// LS Electric XG5000 project: X3353 JOSUNG UPDATE
// PLC NewPLC
// module base 0 slot 0: Motion Module:XGF-M32E (EtherCAT Network, 32-Axis)
// module base 0 slot 1: Input Module:XGI-D28A/B (DC 24V Input, 64 Contacts)
// module base 0 slot 2: Input Module:XGI-D28A/B (DC 24V Input, 64 Contacts)
// module base 0 slot 3: Output Module:XGQ-TR8A/B (Transistor Output, 64 Contacts (0.1A, Sink Output/Source Output))
// module base 0 slot 4: Output Module:XGQ-TR8A/B (Transistor Output, 64 Contacts (0.1A, Sink Output/Source Output))
// module base 0 slot 5: Analog Input Module:XGF-AD16A (A/D Voltage/Current Input Type(16 Channels))
// module base 0 slot 6: Analog Input Module:XGF-AD16A (A/D Voltage/Current Input Type(16 Channels))
// module base 0 slot 7: FEnet:XGL-EFMT(B) (Fast Ethernet Module, Electrical Master)
// module base 0 slot 8: FEnet:XGL-EFMT(B) (Fast Ethernet Module, Electrical Master)

PROGRAM 01_MAIN (task: ¨ö¨¬A¥ì CA¡¤I¡¾¡¿¡¤¡Í)

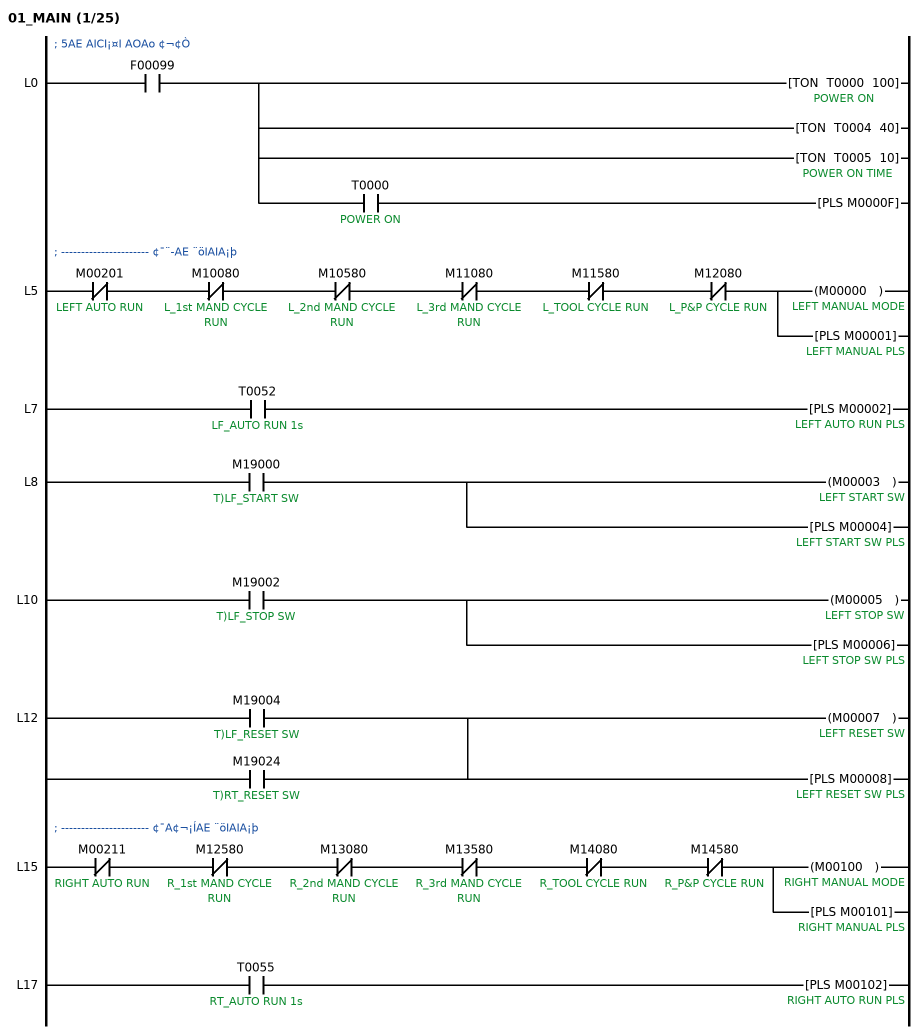
; L0
LOAD      F00099
TON       T0000 100	// POWER ON
TON       T0004 40
TON       T0005 10	// POWER ON TIME
AND       T0000	// POWER ON
OUTP      M0000F
// output comment: 5AE AICI¡¤I AOAo ¢¬¢Ò
// ---------------------- ¢¯¨­AE ¨öIAIA¡þ
; L5
LOAD NOT  M00201	// LEFT AUTO RUN
AND NOT   M10080	// L_1st MAND CYCLE RUN
AND NOT   M10580	// L_2nd MAND CYCLE RUN
AND NOT   M11080	// L_3rd MAND CYCLE RUN
AND NOT   M11580	// L_TOOL CYCLE RUN
AND NOT   M12080	// L_P&P CYCLE RUN
OUT       M00000	// LEFT MANUAL MODE
OUTP      M00001	// LEFT MANUAL PLS
; L7
LOAD      T0052	// LF_AUTO RUN 1s
OUTP      M00002	// LEFT AUTO RUN PLS
; L8
LOAD      M19000	// T)LF_START SW
OUT       M00003	// LEFT START SW
OUTP      M00004	// LEFT START SW PLS
; L10
LOAD      M19002	// T)LF_STOP SW
OUT       M00005	// LEFT STOP SW
OUTP      M00006	// LEFT STOP SW PLS
; L12
LOAD      M19004	// T)LF_RESET SW
OR        M19024	// T)RT_RESET SW
OUT       M00007	// LEFT RESET SW
OUTP      M00008	// LEFT RESET SW PLS
// ---------------------- ¢¯A¢¬¡ÍAE ¨öIAIA¡þ
; L15
LOAD NOT  M00211	// RIGHT AUTO RUN
AND NOT   M12580	// R_1st MAND CYCLE RUN
AND NOT   M13080	// R_2nd MAND CYCLE RUN
AND NOT   M13580	// R_3rd MAND CYCLE RUN
AND NOT   M14080	// R_TOOL CYCLE RUN
AND NOT   M14580	// R_P&P CYCLE RUN
OUT       M00100	// RIGHT MANUAL MODE
OUTP      M00101	// RIGHT MANUAL PLS
; L17
LOAD      T0055	// RT_AUTO RUN 1s
OUTP      M00102	// RIGHT AUTO RUN PLS

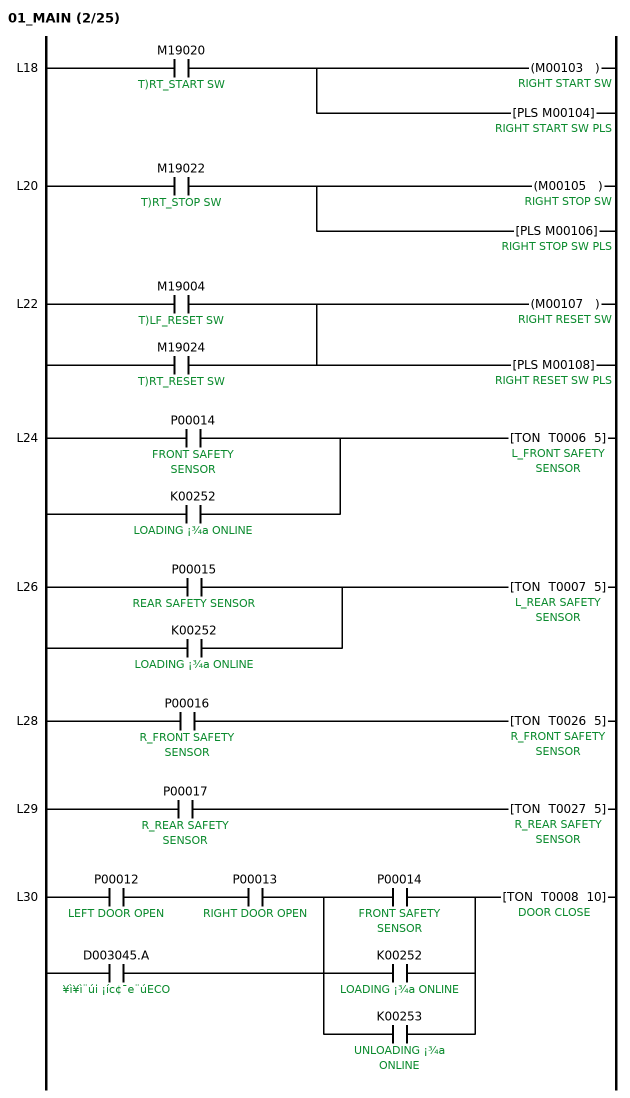
; L18
LOAD      M19020	// T)RT_START SW
OUT       M00103	// RIGHT START SW
OUTP      M00104	// RIGHT START SW PLS
; L20
LOAD      M19022	// T)RT_STOP SW
OUT       M00105	// RIGHT STOP SW
OUTP      M00106	// RIGHT STOP SW PLS
; L22
LOAD      M19004	// T)LF_RESET SW
OR        M19024	// T)RT_RESET SW
OUT       M00107	// RIGHT RESET SW
OUTP      M00108	// RIGHT RESET SW PLS
; L24
LOAD      P00014	// FRONT SAFETY SENSOR
OR        K00252	// LOADING ¡¾a ONLINE
TON       T0006 5	// L_FRONT SAFETY SENSOR
; L26
LOAD      P00015	// REAR SAFETY SENSOR
OR        K00252	// LOADING ¡¾a ONLINE
TON       T0007 5	// L_REAR SAFETY SENSOR
; L28
LOAD      P00016	// R_FRONT SAFETY SENSOR
TON       T0026 5	// R_FRONT SAFETY SENSOR
; L29
LOAD      P00017	// R_REAR SAFETY SENSOR
TON       T0027 5	// R_REAR SAFETY SENSOR
; L30
LOAD      P00012	// LEFT DOOR OPEN
AND       P00013	// RIGHT DOOR OPEN
OR        D003045.A	// ¥ì¥ì¨úi ¡íc¢¯e¨úECO
LOAD      P00014	// FRONT SAFETY SENSOR
OR        K00252	// LOADING ¡¾a ONLINE
OR        K00253	// UNLOADING ¡¾a ONLINE
AND LOAD
TON       T0008 10	// DOOR CLOSE

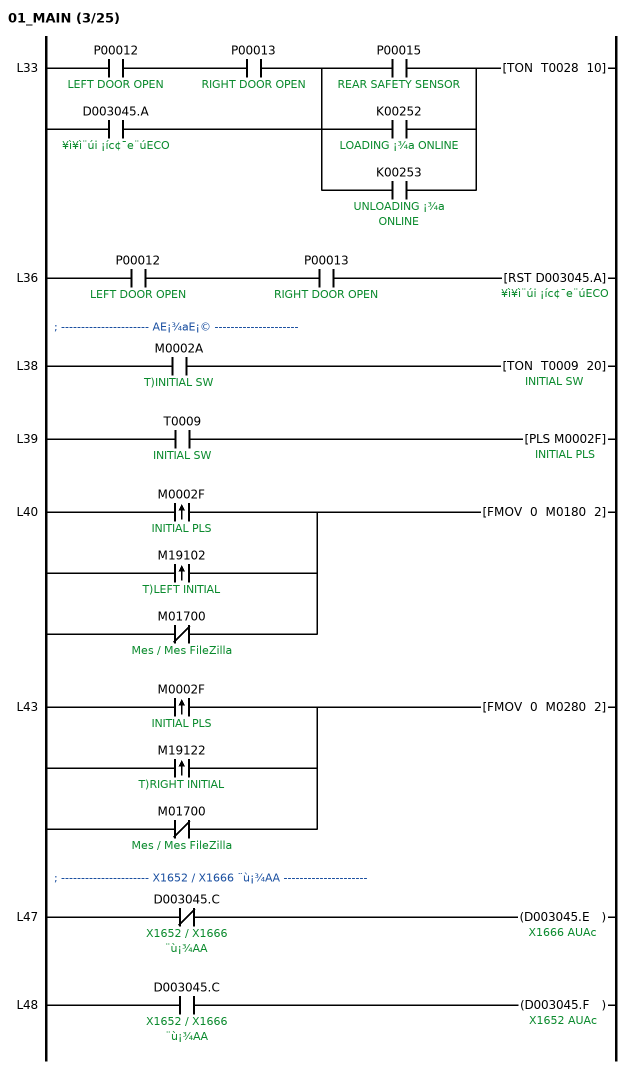
; L33
LOAD      P00012	// LEFT DOOR OPEN
AND       P00013	// RIGHT DOOR OPEN
OR        D003045.A	// ¥ì¥ì¨úi ¡íc¢¯e¨úECO
LOAD      P00015	// REAR SAFETY SENSOR
OR        K00252	// LOADING ¡¾a ONLINE
OR        K00253	// UNLOADING ¡¾a ONLINE
AND LOAD
TON       T0028 10
; L36
LOAD      P00012	// LEFT DOOR OPEN
AND       P00013	// RIGHT DOOR OPEN
RST       D003045.A	// ¥ì¥ì¨úi ¡íc¢¯e¨úECO
// ---------------------- AE¡¾aE¡© ---------------------
; L38
LOAD      M0002A	// T)INITIAL SW
TON       T0009 20	// INITIAL SW
; L39
LOAD      T0009	// INITIAL SW
OUTP      M0002F	// INITIAL PLS
; L40
LOADP     M0002F	// INITIAL PLS
ORP       M19102	// T)LEFT INITIAL
OR NOT    M01700	// Mes / Mes FileZilla
FMOV      0 M0180 2
; L43
LOADP     M0002F	// INITIAL PLS
ORP       M19122	// T)RIGHT INITIAL
OR NOT    M01700	// Mes / Mes FileZilla
FMOV      0 M0280 2
// ---------------------- X1652 / X1666 ¨ù¡¾AA ---------------------
; L47
LOAD NOT  D003045.C	// X1652 / X1666 ¨ù¡¾AA
OUT       D003045.E	// X1666 AUAc
; L48
LOAD      D003045.C	// X1652 / X1666 ¨ù¡¾AA
OUT       D003045.F	// X1652 AUAc

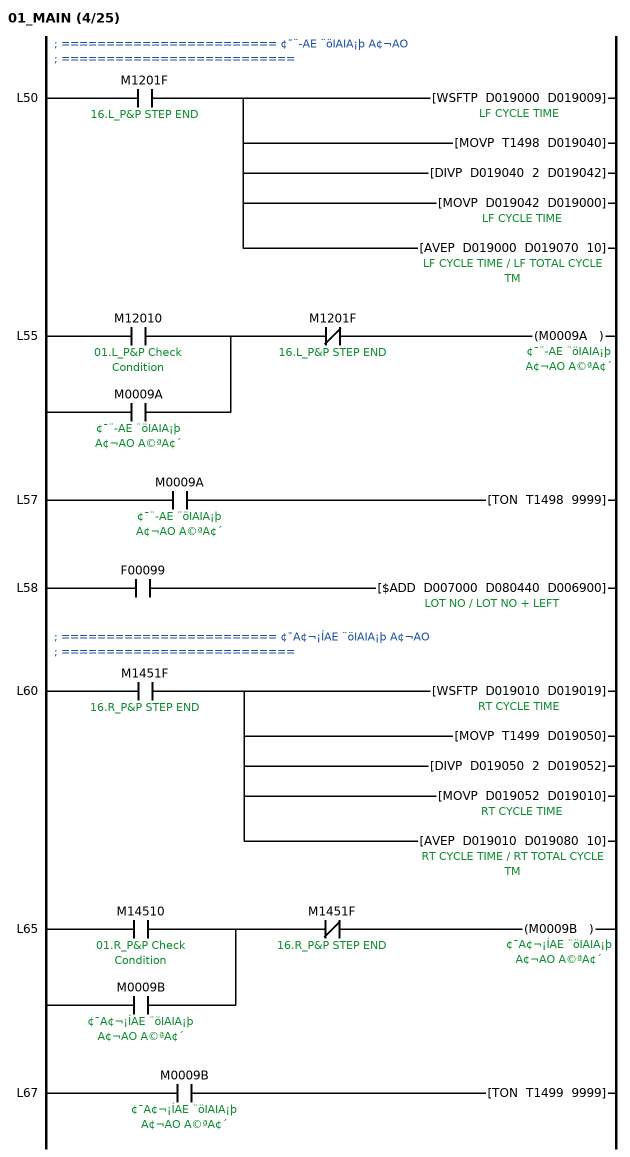
// ======================== ¢¯¨­AE ¨öIAIA¡þ A¢¬AO ==========================
; L50
LOAD      M1201F	// 16.L_P&P STEP END
WSFTP     D019000 D019009	// LF CYCLE TIME
MOVP      T1498 D019040
DIVP      D019040 2 D019042
MOVP      D019042 D019000	// LF CYCLE TIME
AVEP      D019000 D019070 10	// LF CYCLE TIME / LF TOTAL CYCLE TM
; L55
LOAD      M12010	// 01.L_P&P Check Condition
OR        M0009A	// ¢¯¨­AE ¨öIAIA¡þ A¢¬AO A©ªA¢´
AND NOT   M1201F	// 16.L_P&P STEP END
OUT       M0009A	// ¢¯¨­AE ¨öIAIA¡þ A¢¬AO A©ªA¢´
; L57
LOAD      M0009A	// ¢¯¨­AE ¨öIAIA¡þ A¢¬AO A©ªA¢´
TON       T1498 9999
; L58
LOAD      F00099
$ADD      D007000 D080440 D006900	// LOT NO / LOT NO + LEFT
// ======================== ¢¯A¢¬¡ÍAE ¨öIAIA¡þ A¢¬AO ==========================
; L60
LOAD      M1451F	// 16.R_P&P STEP END
WSFTP     D019010 D019019	// RT CYCLE TIME
MOVP      T1499 D019050
DIVP      D019050 2 D019052
MOVP      D019052 D019010	// RT CYCLE TIME
AVEP      D019010 D019080 10	// RT CYCLE TIME / RT TOTAL CYCLE TM
; L65
LOAD      M14510	// 01.R_P&P Check Condition
OR        M0009B	// ¢¯A¢¬¡ÍAE ¨öIAIA¡þ A¢¬AO A©ªA¢´
AND NOT   M1451F	// 16.R_P&P STEP END
OUT       M0009B	// ¢¯A¢¬¡ÍAE ¨öIAIA¡þ A¢¬AO A©ªA¢´
; L67
LOAD      M0009B	// ¢¯A¢¬¡ÍAE ¨öIAIA¡þ A¢¬AO A©ªA¢´
TON       T1499 9999

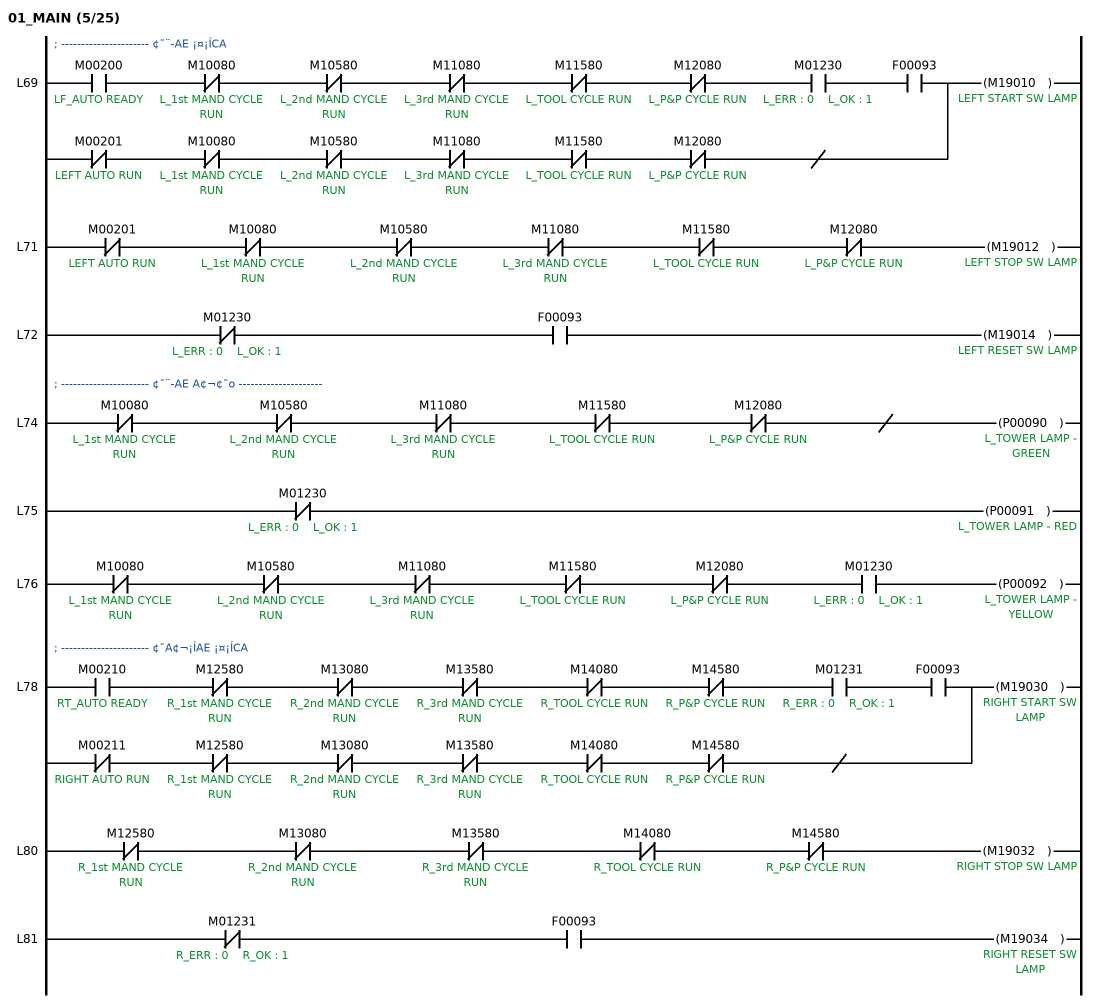
// ---------------------- ¢¯¨­AE ¡¤¡ÍCA
; L69
LOAD      M00200	// LF_AUTO READY
AND NOT   M10080	// L_1st MAND CYCLE RUN
AND NOT   M10580	// L_2nd MAND CYCLE RUN
AND NOT   M11080	// L_3rd MAND CYCLE RUN
AND NOT   M11580	// L_TOOL CYCLE RUN
AND NOT   M12080	// L_P&P CYCLE RUN
AND       M01230	// L_ERR : 0    L_OK : 1
AND       F00093
LOAD NOT  M00201	// LEFT AUTO RUN
AND NOT   M10080	// L_1st MAND CYCLE RUN
AND NOT   M10580	// L_2nd MAND CYCLE RUN
AND NOT   M11080	// L_3rd MAND CYCLE RUN
AND NOT   M11580	// L_TOOL CYCLE RUN
AND NOT   M12080	// L_P&P CYCLE RUN
NOT
OR LOAD
OUT       M19010	// LEFT START SW LAMP
; L71
LOAD NOT  M00201	// LEFT AUTO RUN
AND NOT   M10080	// L_1st MAND CYCLE RUN
AND NOT   M10580	// L_2nd MAND CYCLE RUN
AND NOT   M11080	// L_3rd MAND CYCLE RUN
AND NOT   M11580	// L_TOOL CYCLE RUN
AND NOT   M12080	// L_P&P CYCLE RUN
OUT       M19012	// LEFT STOP SW LAMP
; L72
LOAD NOT  M01230	// L_ERR : 0    L_OK : 1
AND       F00093
OUT       M19014	// LEFT RESET SW LAMP
// ---------------------- ¢¯¨­AE A¢¬¢¯o ---------------------
; L74
LOAD NOT  M10080	// L_1st MAND CYCLE RUN
AND NOT   M10580	// L_2nd MAND CYCLE RUN
AND NOT   M11080	// L_3rd MAND CYCLE RUN
AND NOT   M11580	// L_TOOL CYCLE RUN
AND NOT   M12080	// L_P&P CYCLE RUN
NOT
OUT       P00090	// L_TOWER LAMP - GREEN
; L75
LOAD NOT  M01230	// L_ERR : 0    L_OK : 1
OUT       P00091	// L_TOWER LAMP - RED
; L76
LOAD NOT  M10080	// L_1st MAND CYCLE RUN
AND NOT   M10580	// L_2nd MAND CYCLE RUN
AND NOT   M11080	// L_3rd MAND CYCLE RUN
AND NOT   M11580	// L_TOOL CYCLE RUN
AND NOT   M12080	// L_P&P CYCLE RUN
AND       M01230	// L_ERR : 0    L_OK : 1
OUT       P00092	// L_TOWER LAMP - YELLOW
// ---------------------- ¢¯A¢¬¡ÍAE ¡¤¡ÍCA
; L78
LOAD      M00210	// RT_AUTO READY
AND NOT   M12580	// R_1st MAND CYCLE RUN
AND NOT   M13080	// R_2nd MAND CYCLE RUN
AND NOT   M13580	// R_3rd MAND CYCLE RUN
AND NOT   M14080	// R_TOOL CYCLE RUN
AND NOT   M14580	// R_P&P CYCLE RUN
AND       M01231	// R_ERR : 0    R_OK : 1
AND       F00093
LOAD NOT  M00211	// RIGHT AUTO RUN
AND NOT   M12580	// R_1st MAND CYCLE RUN
AND NOT   M13080	// R_2nd MAND CYCLE RUN
AND NOT   M13580	// R_3rd MAND CYCLE RUN
AND NOT   M14080	// R_TOOL CYCLE RUN
AND NOT   M14580	// R_P&P CYCLE RUN
NOT
OR LOAD
OUT       M19030	// RIGHT START SW LAMP
; L80
LOAD NOT  M12580	// R_1st MAND CYCLE RUN
AND NOT   M13080	// R_2nd MAND CYCLE RUN
AND NOT   M13580	// R_3rd MAND CYCLE RUN
AND NOT   M14080	// R_TOOL CYCLE RUN
AND NOT   M14580	// R_P&P CYCLE RUN
OUT       M19032	// RIGHT STOP SW LAMP
; L81
LOAD NOT  M01231	// R_ERR : 0    R_OK : 1
AND       F00093
OUT       M19034	// RIGHT RESET SW LAMP

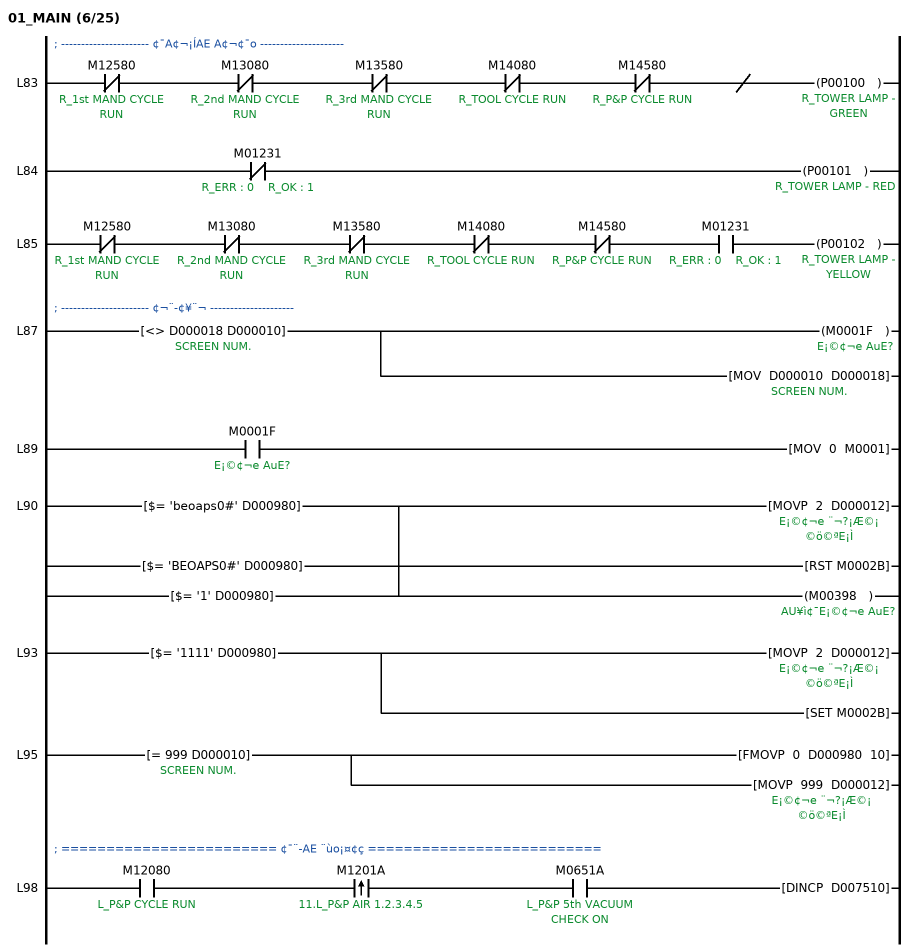
// ---------------------- ¢¯A¢¬¡ÍAE A¢¬¢¯o ---------------------
; L83
LOAD NOT  M12580	// R_1st MAND CYCLE RUN
AND NOT   M13080	// R_2nd MAND CYCLE RUN
AND NOT   M13580	// R_3rd MAND CYCLE RUN
AND NOT   M14080	// R_TOOL CYCLE RUN
AND NOT   M14580	// R_P&P CYCLE RUN
NOT
OUT       P00100	// R_TOWER LAMP - GREEN
; L84
LOAD NOT  M01231	// R_ERR : 0    R_OK : 1
OUT       P00101	// R_TOWER LAMP - RED
; L85
LOAD NOT  M12580	// R_1st MAND CYCLE RUN
AND NOT   M13080	// R_2nd MAND CYCLE RUN
AND NOT   M13580	// R_3rd MAND CYCLE RUN
AND NOT   M14080	// R_TOOL CYCLE RUN
AND NOT   M14580	// R_P&P CYCLE RUN
AND       M01231	// R_ERR : 0    R_OK : 1
OUT       P00102	// R_TOWER LAMP - YELLOW
// ---------------------- ¢¬¨­¢¥¨¬ ---------------------
; L87
LOAD<>    D000018 D000010	// SCREEN NUM.
OUT       M0001F	// E¡©¢¬e AuE?
MOV       D000010 D000018	// SCREEN NUM.
; L89
LOAD      M0001F	// E¡©¢¬e AuE?
MOV       0 M0001
; L90
LOAD$=    'beoaps0#' D000980
OR$=      'BEOAPS0#' D000980
OR$=      '1' D000980
MOVP      2 D000012	// E¡©¢¬e ¨¬?¡Æ©¡ ©ö©ªE¡Ì
RST       M0002B
OUT       M00398	// AU¥ì¢¯E¡©¢¬e AuE?
; L93
LOAD$=    '1111' D000980
MOVP      2 D000012	// E¡©¢¬e ¨¬?¡Æ©¡ ©ö©ªE¡Ì
SET       M0002B
; L95
LOAD=     999 D000010	// SCREEN NUM.
FMOVP     0 D000980 10
MOVP      999 D000012	// E¡©¢¬e ¨¬?¡Æ©¡ ©ö©ªE¡Ì
// ======================== ¢¯¨­AE ¨ùo¡¤¢ç ==========================
; L98
LOAD      M12080	// L_P&P CYCLE RUN
ANDP      M1201A	// 11.L_P&P AIR 1.2.3.4.5
AND       M0651A	// L_P&P 5th VACUUM CHECK ON
DINCP     D007510

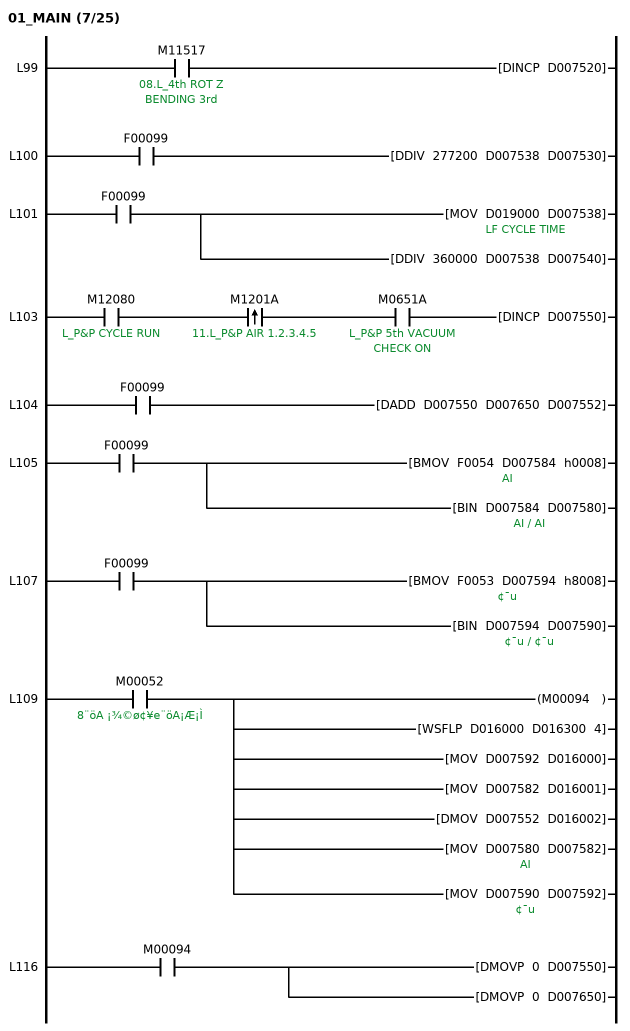
; L99
LOAD      M11517	// 08.L_4th ROT Z BENDING 3rd
DINCP     D007520
; L100
LOAD      F00099
DDIV      277200 D007538 D007530
; L101
LOAD      F00099
MOV       D019000 D007538	// LF CYCLE TIME
DDIV      360000 D007538 D007540
; L103
LOAD      M12080	// L_P&P CYCLE RUN
ANDP      M1201A	// 11.L_P&P AIR 1.2.3.4.5
AND       M0651A	// L_P&P 5th VACUUM CHECK ON
DINCP     D007550
; L104
LOAD      F00099
DADD      D007550 D007650 D007552
; L105
LOAD      F00099
BMOV      F0054 D007584 h0008	// AI
BIN       D007584 D007580	// AI / AI
; L107
LOAD      F00099
BMOV      F0053 D007594 h8008	// ¢¯u
BIN       D007594 D007590	// ¢¯u / ¢¯u
; L109
LOAD      M00052	// 8¨öA ¡¾©ø¢¥e¨öA¡Æ¡Ì
OUT       M00094
WSFLP     D016000 D016300 4
MOV       D007592 D016000
MOV       D007582 D016001
DMOV      D007552 D016002
MOV       D007580 D007582	// AI
MOV       D007590 D007592	// ¢¯u
; L116
LOAD      M00094
DMOVP     0 D007550
DMOVP     0 D007650

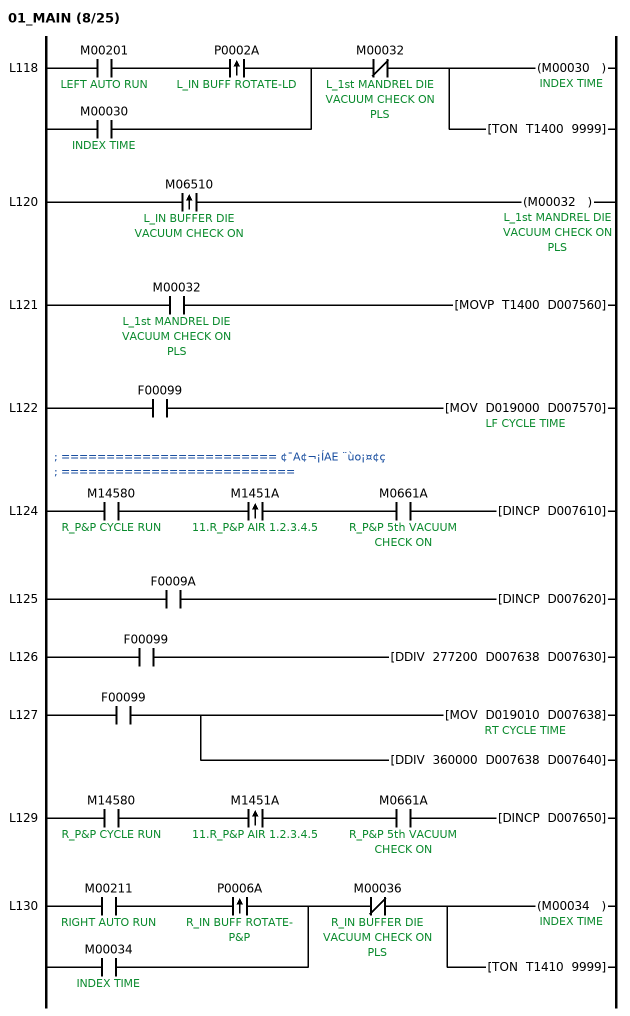
; L118
LOAD      M00201	// LEFT AUTO RUN
ANDP      P0002A	// L_IN BUFF ROTATE-LD
OR        M00030	// INDEX TIME
AND NOT   M00032	// L_1st MANDREL DIE VACUUM CHECK ON PLS
OUT       M00030	// INDEX TIME
TON       T1400 9999
; L120
LOADP     M06510	// L_IN BUFFER DIE VACUUM CHECK ON
OUT       M00032	// L_1st MANDREL DIE VACUUM CHECK ON PLS
; L121
LOAD      M00032	// L_1st MANDREL DIE VACUUM CHECK ON PLS
MOVP      T1400 D007560
; L122
LOAD      F00099
MOV       D019000 D007570	// LF CYCLE TIME
// ======================== ¢¯A¢¬¡ÍAE ¨ùo¡¤¢ç ==========================
; L124
LOAD      M14580	// R_P&P CYCLE RUN
ANDP      M1451A	// 11.R_P&P AIR 1.2.3.4.5
AND       M0661A	// R_P&P 5th VACUUM CHECK ON
DINCP     D007610
; L125
LOAD      F0009A
DINCP     D007620
; L126
LOAD      F00099
DDIV      277200 D007638 D007630
; L127
LOAD      F00099
MOV       D019010 D007638	// RT CYCLE TIME
DDIV      360000 D007638 D007640
; L129
LOAD      M14580	// R_P&P CYCLE RUN
ANDP      M1451A	// 11.R_P&P AIR 1.2.3.4.5
AND       M0661A	// R_P&P 5th VACUUM CHECK ON
DINCP     D007650
; L130
LOAD      M00211	// RIGHT AUTO RUN
ANDP      P0006A	// R_IN BUFF ROTATE- P&P
OR        M00034	// INDEX TIME
AND NOT   M00036	// R_IN BUFFER DIE VACUUM CHECK ON PLS
OUT       M00034	// INDEX TIME
TON       T1410 9999

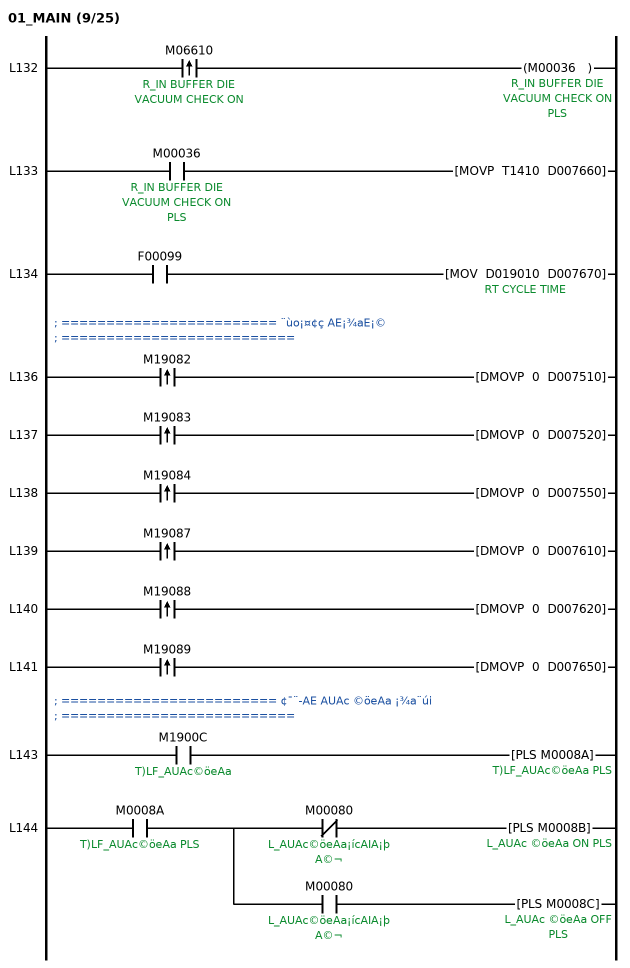
; L132
LOADP     M06610	// R_IN BUFFER DIE VACUUM CHECK ON
OUT       M00036	// R_IN BUFFER DIE VACUUM CHECK ON PLS
; L133
LOAD      M00036	// R_IN BUFFER DIE VACUUM CHECK ON PLS
MOVP      T1410 D007660
; L134
LOAD      F00099
MOV       D019010 D007670	// RT CYCLE TIME
// ======================== ¨ùo¡¤¢ç AE¡¾aE¡© ==========================
; L136
LOADP     M19082
DMOVP     0 D007510
; L137
LOADP     M19083
DMOVP     0 D007520
; L138
LOADP     M19084
DMOVP     0 D007550
; L139
LOADP     M19087
DMOVP     0 D007610
; L140
LOADP     M19088
DMOVP     0 D007620
; L141
LOADP     M19089
DMOVP     0 D007650
// ======================== ¢¯¨­AE AUAc ©öeAa ¡¾a¨úi ==========================
; L143
LOAD      M1900C	// T)LF_AUAc©öeAa
OUTP      M0008A	// T)LF_AUAc©öeAa PLS
; L144
LOAD      M0008A	// T)LF_AUAc©öeAa PLS
MPUSH
AND NOT   M00080	// L_AUAc©öeAa¡ícAIA¡þA©¬
OUTP      M0008B	// L_AUAc ©öeAa ON PLS
MPOP
AND       M00080	// L_AUAc©öeAa¡ícAIA¡þA©¬
OUTP      M0008C	// L_AUAc ©öeAa OFF PLS

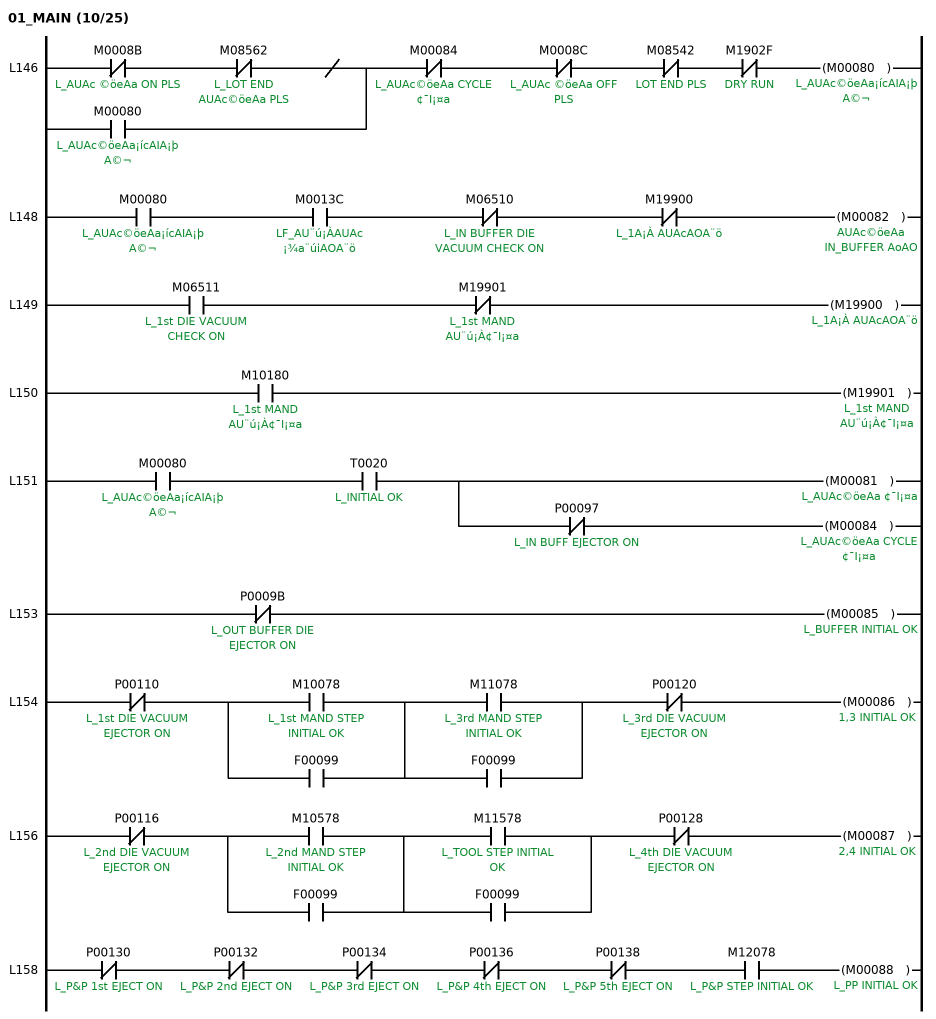
; L146
LOAD NOT  M0008B	// L_AUAc ©öeAa ON PLS
AND NOT   M08562	// L_LOT END AUAc©öeAa PLS
NOT
OR        M00080	// L_AUAc©öeAa¡ícAIA¡þA©¬
AND NOT   M00084	// L_AUAc©öeAa CYCLE ¢¯I¡¤a
AND NOT   M0008C	// L_AUAc ©öeAa OFF PLS
AND NOT   M08542	// LOT END PLS
AND NOT   M1902F	// DRY RUN
OUT       M00080	// L_AUAc©öeAa¡ícAIA¡þA©¬
; L148
LOAD      M00080	// L_AUAc©öeAa¡ícAIA¡þA©¬
AND       M0013C	// LF_AU¨ú¡ÀAUAc ¡¾a¨úiAOA¨ö
AND NOT   M06510	// L_IN BUFFER DIE VACUUM CHECK ON
AND NOT   M19900	// L_1A¡À AUAcAOA¨ö
OUT       M00082	// AUAc©öeAa IN_BUFFER AoAO 
; L149
LOAD      M06511	// L_1st DIE VACUUM CHECK ON
AND NOT   M19901	// L_1st MAND AU¨ú¡À¢¯I¡¤a
OUT       M19900	// L_1A¡À AUAcAOA¨ö
; L150
LOAD      M10180	// L_1st MAND AU¨ú¡À¢¯I¡¤a
OUT       M19901	// L_1st MAND AU¨ú¡À¢¯I¡¤a
; L151
LOAD      M00080	// L_AUAc©öeAa¡ícAIA¡þA©¬
AND       T0020	// L_INITIAL OK
OUT       M00081	// L_AUAc©öeAa ¢¯I¡¤a
AND NOT   P00097	// L_IN BUFF EJECTOR ON
OUT       M00084	// L_AUAc©öeAa CYCLE ¢¯I¡¤a
; L153
LOAD NOT  P0009B	// L_OUT BUFFER DIE EJECTOR ON
OUT       M00085	// L_BUFFER INITIAL OK
; L154
LOAD NOT  P00110	// L_1st DIE VACUUM EJECTOR ON
LOAD      M10078	// L_1st MAND STEP INITIAL OK
OR        F00099
AND LOAD
LOAD      M11078	// L_3rd MAND STEP INITIAL OK
OR        F00099
AND LOAD
AND NOT   P00120	// L_3rd DIE VACUUM EJECTOR ON
OUT       M00086	// 1,3 INITIAL OK
; L156
LOAD NOT  P00116	// L_2nd DIE VACUUM EJECTOR ON
LOAD      M10578	// L_2nd MAND STEP INITIAL OK
OR        F00099
AND LOAD
LOAD      M11578	// L_TOOL STEP INITIAL OK
OR        F00099
AND LOAD
AND NOT   P00128	// L_4th DIE VACUUM EJECTOR ON
OUT       M00087	// 2,4 INITIAL OK
; L158
LOAD NOT  P00130	// L_P&P 1st EJECT ON
AND NOT   P00132	// L_P&P 2nd EJECT ON
AND NOT   P00134	// L_P&P 3rd EJECT ON
AND NOT   P00136	// L_P&P 4th EJECT ON
AND NOT   P00138	// L_P&P 5th EJECT ON
AND       M12078	// L_P&P STEP INITIAL OK
OUT       M00088	// L_PP INITIAL OK

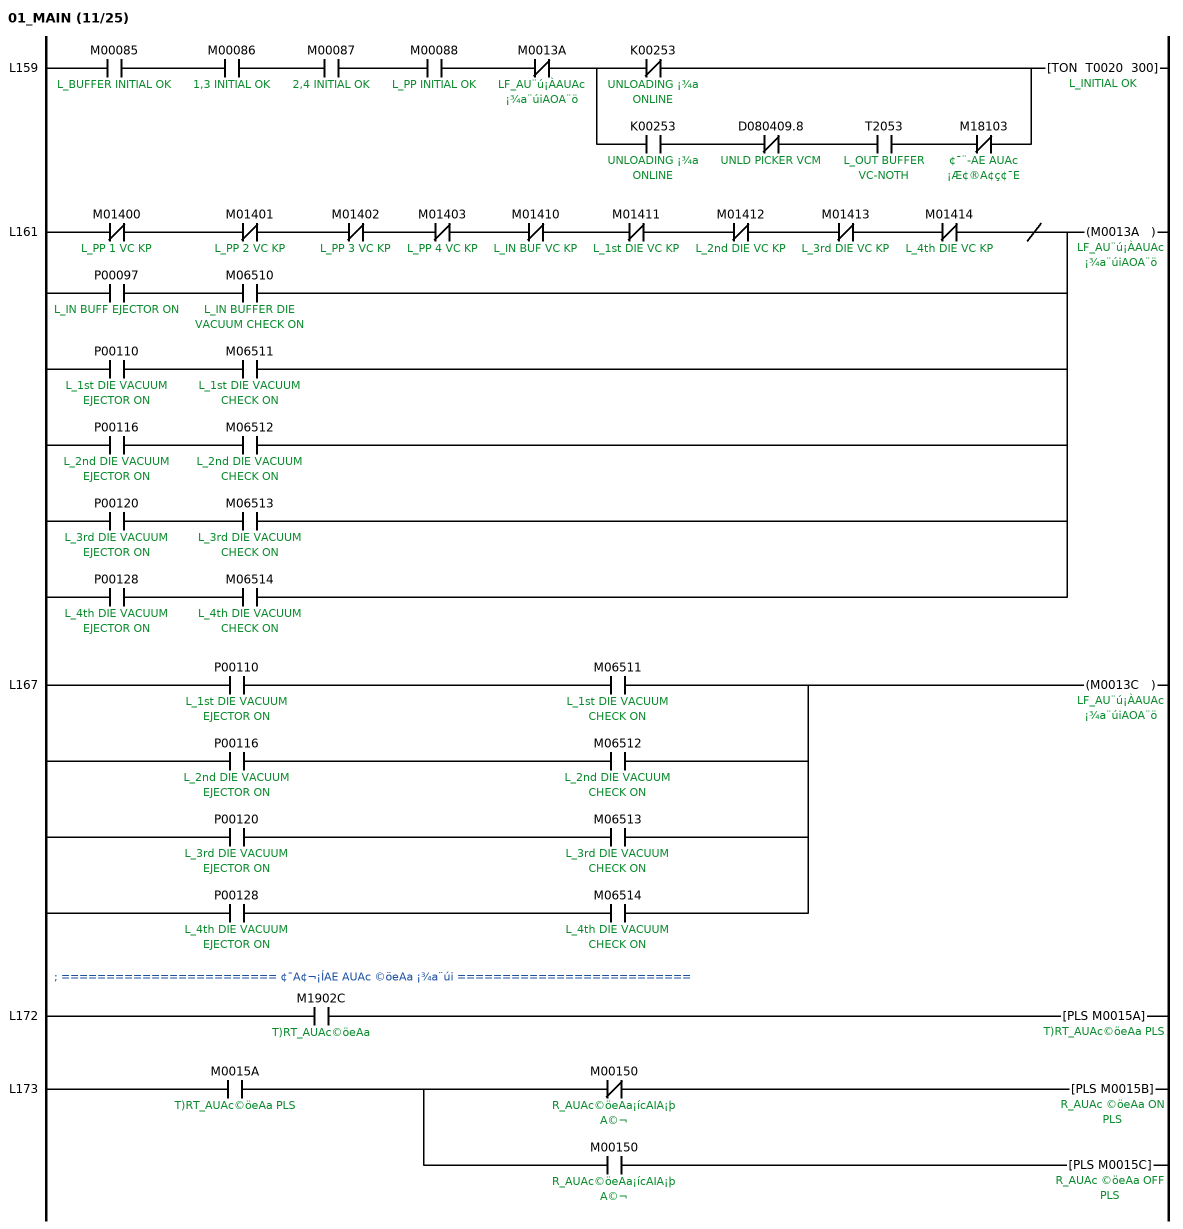
; L159
LOAD      M00085	// L_BUFFER INITIAL OK
AND       M00086	// 1,3 INITIAL OK
AND       M00087	// 2,4 INITIAL OK
AND       M00088	// L_PP INITIAL OK
AND NOT   M0013A	// LF_AU¨ú¡ÀAUAc ¡¾a¨úiAOA¨ö
LOAD NOT  K00253	// UNLOADING ¡¾a ONLINE
LOAD      K00253	// UNLOADING ¡¾a ONLINE
AND NOT   D080409.8	// UNLD PICKER VCM
AND       T2053	// L_OUT BUFFER VC-NOTH
AND NOT   M18103	// ¢¯¨­AE AUAc ¡Æ¢®A¢ç¢¯E
OR LOAD
AND LOAD
TON       T0020 300	// L_INITIAL OK
; L161
LOAD NOT  M01400	// L_PP 1 VC KP
AND NOT   M01401	// L_PP 2 VC KP
AND NOT   M01402	// L_PP 3 VC KP
AND NOT   M01403	// L_PP 4 VC KP
AND NOT   M01410	// L_IN BUF VC KP
AND NOT   M01411	// L_1st DIE VC KP
AND NOT   M01412	// L_2nd DIE VC KP
AND NOT   M01413	// L_3rd DIE VC KP
AND NOT   M01414	// L_4th DIE VC KP
NOT
LOAD      P00097	// L_IN BUFF EJECTOR ON
AND       M06510	// L_IN BUFFER DIE VACUUM CHECK ON
OR LOAD
LOAD      P00110	// L_1st DIE VACUUM EJECTOR ON
AND       M06511	// L_1st DIE VACUUM CHECK ON
OR LOAD
LOAD      P00116	// L_2nd DIE VACUUM EJECTOR ON
AND       M06512	// L_2nd DIE VACUUM CHECK ON
OR LOAD
LOAD      P00120	// L_3rd DIE VACUUM EJECTOR ON
AND       M06513	// L_3rd DIE VACUUM CHECK ON
OR LOAD
LOAD      P00128	// L_4th DIE VACUUM EJECTOR ON
AND       M06514	// L_4th DIE VACUUM CHECK ON
OR LOAD
OUT       M0013A	// LF_AU¨ú¡ÀAUAc ¡¾a¨úiAOA¨ö
; L167
LOAD      P00110	// L_1st DIE VACUUM EJECTOR ON
AND       M06511	// L_1st DIE VACUUM CHECK ON
LOAD      P00116	// L_2nd DIE VACUUM EJECTOR ON
AND       M06512	// L_2nd DIE VACUUM CHECK ON
OR LOAD
LOAD      P00120	// L_3rd DIE VACUUM EJECTOR ON
AND       M06513	// L_3rd DIE VACUUM CHECK ON
OR LOAD
LOAD      P00128	// L_4th DIE VACUUM EJECTOR ON
AND       M06514	// L_4th DIE VACUUM CHECK ON
OR LOAD
OUT       M0013C	// LF_AU¨ú¡ÀAUAc ¡¾a¨úiAOA¨ö
// ======================== ¢¯A¢¬¡ÍAE AUAc ©öeAa ¡¾a¨úi ==========================
; L172
LOAD      M1902C	// T)RT_AUAc©öeAa
OUTP      M0015A	// T)RT_AUAc©öeAa PLS
; L173
LOAD      M0015A	// T)RT_AUAc©öeAa PLS
MPUSH
AND NOT   M00150	// R_AUAc©öeAa¡ícAIA¡þA©¬
OUTP      M0015B	// R_AUAc ©öeAa ON PLS
MPOP
AND       M00150	// R_AUAc©öeAa¡ícAIA¡þA©¬
OUTP      M0015C	// R_AUAc ©öeAa OFF PLS

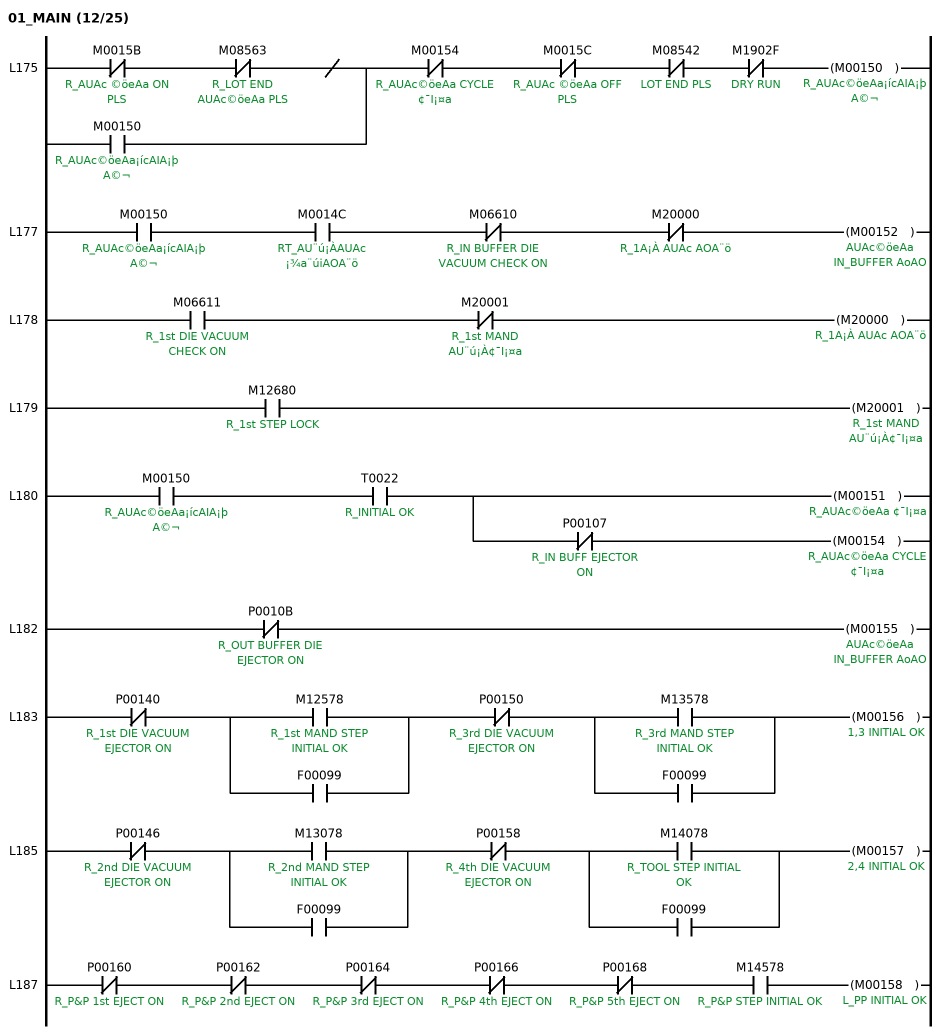
; L175
LOAD NOT  M0015B	// R_AUAc ©öeAa ON PLS
AND NOT   M08563	// R_LOT END AUAc©öeAa PLS
NOT
OR        M00150	// R_AUAc©öeAa¡ícAIA¡þA©¬
AND NOT   M00154	// R_AUAc©öeAa CYCLE ¢¯I¡¤a
AND NOT   M0015C	// R_AUAc ©öeAa OFF PLS
AND NOT   M08542	// LOT END PLS
AND NOT   M1902F	// DRY RUN
OUT       M00150	// R_AUAc©öeAa¡ícAIA¡þA©¬
; L177
LOAD      M00150	// R_AUAc©öeAa¡ícAIA¡þA©¬
AND       M0014C	// RT_AU¨ú¡ÀAUAc ¡¾a¨úiAOA¨ö
AND NOT   M06610	// R_IN BUFFER DIE VACUUM CHECK ON
AND NOT   M20000	// R_1A¡À AUAc AOA¨ö
OUT       M00152	// AUAc©öeAa IN_BUFFER AoAO 
; L178
LOAD      M06611	// R_1st DIE VACUUM CHECK ON
AND NOT   M20001	// R_1st MAND AU¨ú¡À¢¯I¡¤a
OUT       M20000	// R_1A¡À AUAc AOA¨ö
; L179
LOAD      M12680	// R_1st STEP LOCK
OUT       M20001	// R_1st MAND AU¨ú¡À¢¯I¡¤a
; L180
LOAD      M00150	// R_AUAc©öeAa¡ícAIA¡þA©¬
AND       T0022	// R_INITIAL OK
OUT       M00151	// R_AUAc©öeAa ¢¯I¡¤a
AND NOT   P00107	// R_IN BUFF EJECTOR ON
OUT       M00154	// R_AUAc©öeAa CYCLE ¢¯I¡¤a
; L182
LOAD NOT  P0010B	// R_OUT BUFFER DIE EJECTOR ON
OUT       M00155	// AUAc©öeAa IN_BUFFER AoAO 
; L183
LOAD NOT  P00140	// R_1st DIE VACUUM EJECTOR ON
LOAD      M12578	// R_1st MAND STEP INITIAL OK
OR        F00099
AND LOAD
AND NOT   P00150	// R_3rd DIE VACUUM EJECTOR ON
LOAD      M13578	// R_3rd MAND STEP INITIAL OK
OR        F00099
AND LOAD
OUT       M00156	// 1,3 INITIAL OK
; L185
LOAD NOT  P00146	// R_2nd DIE VACUUM EJECTOR ON
LOAD      M13078	// R_2nd MAND STEP INITIAL OK
OR        F00099
AND LOAD
AND NOT   P00158	// R_4th DIE VACUUM EJECTOR ON
LOAD      M14078	// R_TOOL STEP INITIAL OK
OR        F00099
AND LOAD
OUT       M00157	// 2,4 INITIAL OK
; L187
LOAD NOT  P00160	// R_P&P 1st EJECT ON
AND NOT   P00162	// R_P&P 2nd EJECT ON
AND NOT   P00164	// R_P&P 3rd EJECT ON
AND NOT   P00166	// R_P&P 4th EJECT ON
AND NOT   P00168	// R_P&P 5th EJECT ON
AND       M14578	// R_P&P STEP INITIAL OK
OUT       M00158	// L_PP INITIAL OK

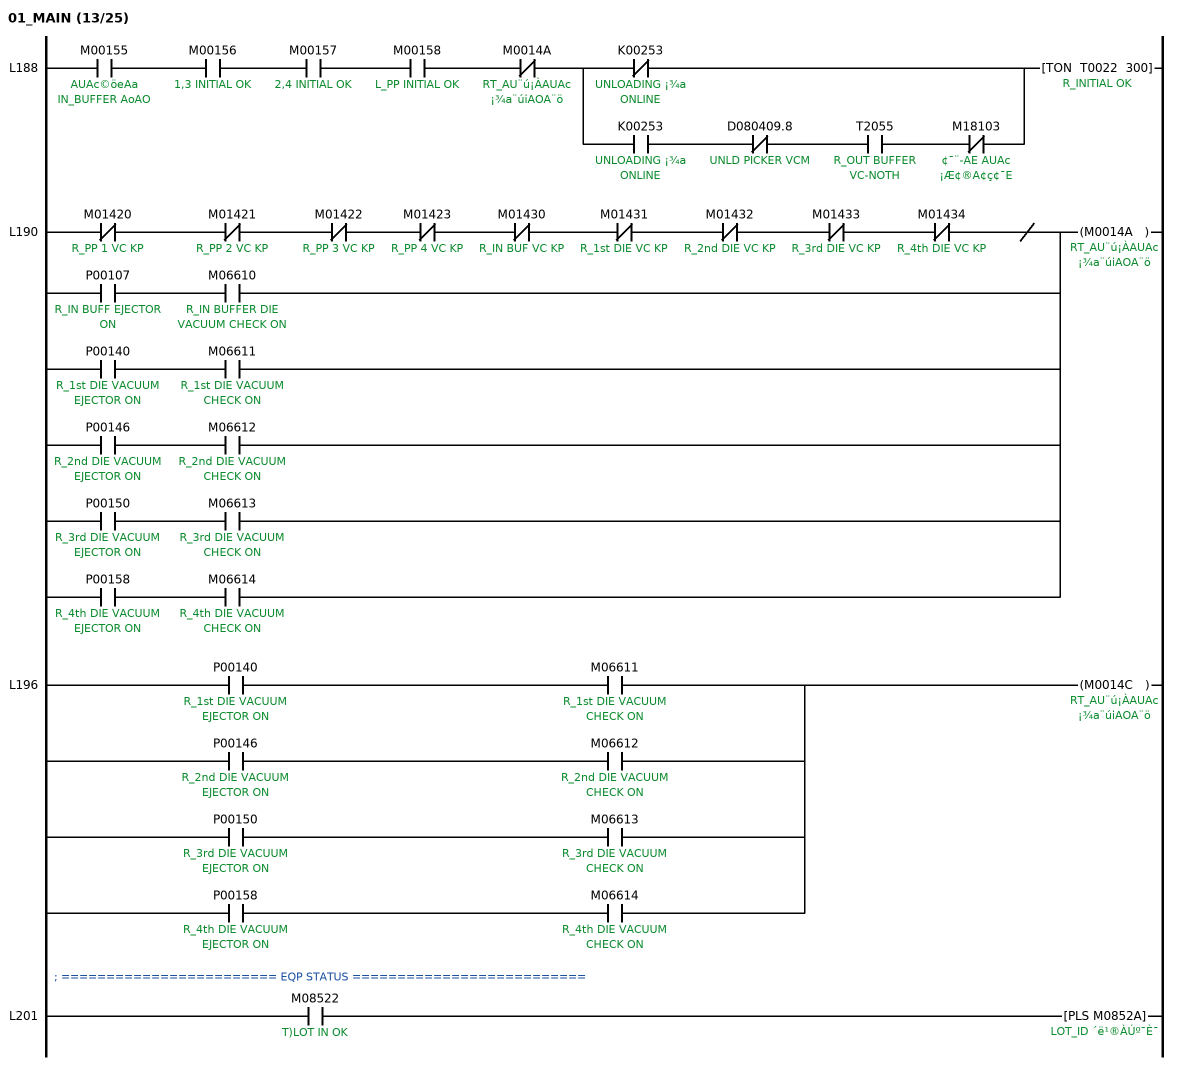
; L188
LOAD      M00155	// AUAc©öeAa IN_BUFFER AoAO 
AND       M00156	// 1,3 INITIAL OK
AND       M00157	// 2,4 INITIAL OK
AND       M00158	// L_PP INITIAL OK
AND NOT   M0014A	// RT_AU¨ú¡ÀAUAc ¡¾a¨úiAOA¨ö
LOAD NOT  K00253	// UNLOADING ¡¾a ONLINE
LOAD      K00253	// UNLOADING ¡¾a ONLINE
AND NOT   D080409.8	// UNLD PICKER VCM
AND       T2055	// R_OUT BUFFER VC-NOTH
AND NOT   M18103	// ¢¯¨­AE AUAc ¡Æ¢®A¢ç¢¯E
OR LOAD
AND LOAD
TON       T0022 300	// R_INITIAL OK
; L190
LOAD NOT  M01420	// R_PP 1 VC KP
AND NOT   M01421	// R_PP 2 VC KP
AND NOT   M01422	// R_PP 3 VC KP
AND NOT   M01423	// R_PP 4 VC KP
AND NOT   M01430	// R_IN BUF VC KP
AND NOT   M01431	// R_1st DIE VC KP
AND NOT   M01432	// R_2nd DIE VC KP
AND NOT   M01433	// R_3rd DIE VC KP
AND NOT   M01434	// R_4th DIE VC KP
NOT
LOAD      P00107	// R_IN BUFF EJECTOR ON
AND       M06610	// R_IN BUFFER DIE VACUUM CHECK ON
OR LOAD
LOAD      P00140	// R_1st DIE VACUUM EJECTOR ON
AND       M06611	// R_1st DIE VACUUM CHECK ON
OR LOAD
LOAD      P00146	// R_2nd DIE VACUUM EJECTOR ON
AND       M06612	// R_2nd DIE VACUUM CHECK ON
OR LOAD
LOAD      P00150	// R_3rd DIE VACUUM EJECTOR ON
AND       M06613	// R_3rd DIE VACUUM CHECK ON
OR LOAD
LOAD      P00158	// R_4th DIE VACUUM EJECTOR ON
AND       M06614	// R_4th DIE VACUUM CHECK ON
OR LOAD
OUT       M0014A	// RT_AU¨ú¡ÀAUAc ¡¾a¨úiAOA¨ö
; L196
LOAD      P00140	// R_1st DIE VACUUM EJECTOR ON
AND       M06611	// R_1st DIE VACUUM CHECK ON
LOAD      P00146	// R_2nd DIE VACUUM EJECTOR ON
AND       M06612	// R_2nd DIE VACUUM CHECK ON
OR LOAD
LOAD      P00150	// R_3rd DIE VACUUM EJECTOR ON
AND       M06613	// R_3rd DIE VACUUM CHECK ON
OR LOAD
LOAD      P00158	// R_4th DIE VACUUM EJECTOR ON
AND       M06614	// R_4th DIE VACUUM CHECK ON
OR LOAD
OUT       M0014C	// RT_AU¨ú¡ÀAUAc ¡¾a¨úiAOA¨ö
// ======================== EQP STATUS ==========================
; L201
LOAD      M08522	// T)LOT IN OK
OUTP      M0852A	// LOT_ID ´ë¹®ÀÚº¯È¯

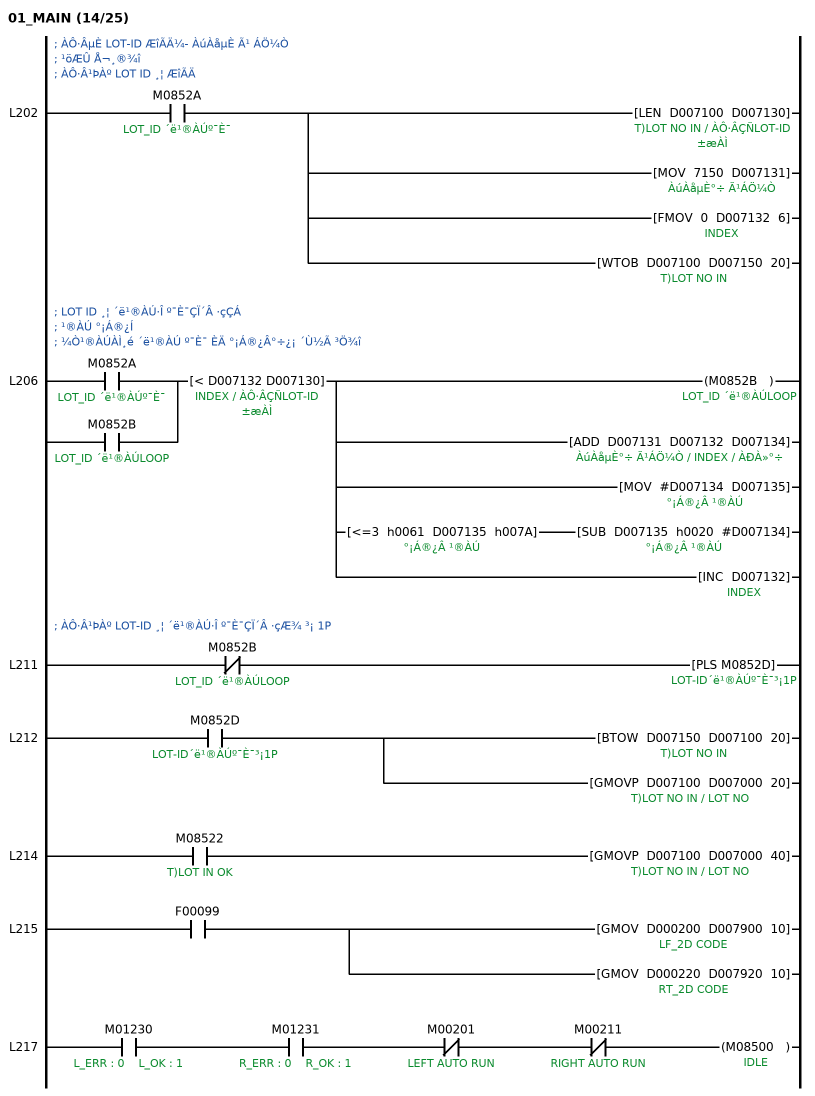
; L202
LOAD      M0852A	// LOT_ID ´ë¹®ÀÚº¯È¯
LEN       D007100 D007130	// T)LOT NO IN / ÀÔ·ÂÇÑLOT-ID ±æÀÌ
MOV       7150 D007131	// ÀúÀåµÈ°÷ Ã¹ÁÖ¼Ò
FMOV      0 D007132 6	// INDEX
WTOB      D007100 D007150 20	// T)LOT NO IN
// output comment: ÀÔ·ÂµÈ LOT-ID ÆîÃÄ¼­ ÀúÀåµÈ Ã¹ ÁÖ¼Ò
// output comment: ¹öÆÛ Å¬¸®¾î
// output comment: ÀÔ·Â¹ÞÀº LOT ID ¸¦ ÆîÃÄ
; L206
LOAD      M0852A	// LOT_ID ´ë¹®ÀÚº¯È¯
OR        M0852B	// LOT_ID ´ë¹®ÀÚLOOP
AND<      D007132 D007130	// INDEX / ÀÔ·ÂÇÑLOT-ID ±æÀÌ
OUT       M0852B	// LOT_ID ´ë¹®ÀÚLOOP
ADD       D007131 D007132 D007134	// ÀúÀåµÈ°÷ Ã¹ÁÖ¼Ò / INDEX / ÀÐÀ»°÷
MOV       #D007134 D007135	// °¡Á®¿Â ¹®ÀÚ
MPUSH
AND<=3    h0061 D007135 h007A	// °¡Á®¿Â ¹®ÀÚ
SUB       D007135 h0020 #D007134	// °¡Á®¿Â ¹®ÀÚ
MPOP
INC       D007132	// INDEX
// output comment: LOT ID ¸¦ ´ë¹®ÀÚ·Î º¯È¯ÇÏ´Â ·çÇÁ
// output comment: ¹®ÀÚ °¡Á®¿Í
// output comment: ¼Ò¹®ÀÚÀÌ¸é ´ë¹®ÀÚ º¯È¯ ÈÄ °¡Á®¿Â°÷¿¡ ´Ù½Ã ³Ö¾î
; L211
LOAD NOT  M0852B	// LOT_ID ´ë¹®ÀÚLOOP
OUTP      M0852D	// LOT-ID´ë¹®ÀÚº¯È¯³¡1P
// output comment: ÀÔ·Â¹ÞÀº LOT-ID ¸¦ ´ë¹®ÀÚ·Î º¯È¯ÇÏ´Â ·çÆ¾ ³¡ 1P
; L212
LOAD      M0852D	// LOT-ID´ë¹®ÀÚº¯È¯³¡1P
BTOW      D007150 D007100 20	// T)LOT NO IN
GMOVP     D007100 D007000 20	// T)LOT NO IN / LOT NO
; L214
LOAD      M08522	// T)LOT IN OK
GMOVP     D007100 D007000 40	// T)LOT NO IN / LOT NO
; L215
LOAD      F00099
GMOV      D000200 D007900 10	// LF_2D CODE
GMOV      D000220 D007920 10	// RT_2D CODE
; L217
LOAD      M01230	// L_ERR : 0    L_OK : 1
AND       M01231	// R_ERR : 0    R_OK : 1
AND NOT   M00201	// LEFT AUTO RUN
AND NOT   M00211	// RIGHT AUTO RUN
OUT       M08500	// IDLE

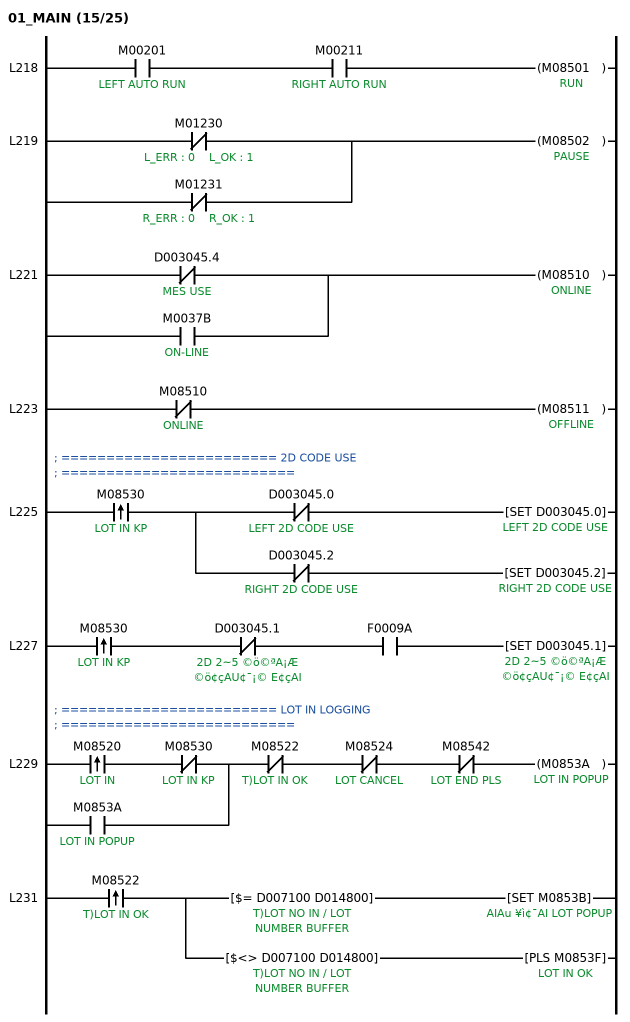
; L218
LOAD      M00201	// LEFT AUTO RUN
AND       M00211	// RIGHT AUTO RUN
OUT       M08501	// RUN
; L219
LOAD NOT  M01230	// L_ERR : 0    L_OK : 1
OR NOT    M01231	// R_ERR : 0    R_OK : 1
OUT       M08502	// PAUSE
; L221
LOAD NOT  D003045.4	// MES USE
OR        M0037B	// ON-LINE
OUT       M08510	// ONLINE
; L223
LOAD NOT  M08510	// ONLINE
OUT       M08511	// OFFLINE
// ======================== 2D CODE USE ==========================
; L225
LOADP     M08530	// LOT IN KP
MPUSH
AND NOT   D003045.0	// LEFT 2D CODE USE
SET       D003045.0	// LEFT 2D CODE USE
MPOP
AND NOT   D003045.2	// RIGHT 2D CODE USE
SET       D003045.2	// RIGHT 2D CODE USE
; L227
LOADP     M08530	// LOT IN KP
AND NOT   D003045.1	// 2D 2~5 ©ö©ªA¡Æ ©ö¢çAU¢¯¡© E¢çAI
AND       F0009A
SET       D003045.1	// 2D 2~5 ©ö©ªA¡Æ ©ö¢çAU¢¯¡© E¢çAI
// ======================== LOT IN LOGGING ==========================
; L229
LOADP     M08520	// LOT IN
AND NOT   M08530	// LOT IN KP
OR        M0853A	// LOT IN POPUP
AND NOT   M08522	// T)LOT IN OK
AND NOT   M08524	// LOT CANCEL
AND NOT   M08542	// LOT END PLS
OUT       M0853A	// LOT IN POPUP
; L231
LOADP     M08522	// T)LOT IN OK
MPUSH
AND$=     D007100 D014800	// T)LOT NO IN / LOT NUMBER BUFFER
SET       M0853B	// AIAu ¥ì¢¯AI LOT POPUP
MPOP
AND$<>    D007100 D014800	// T)LOT NO IN / LOT NUMBER BUFFER
OUTP      M0853F	// LOT IN OK

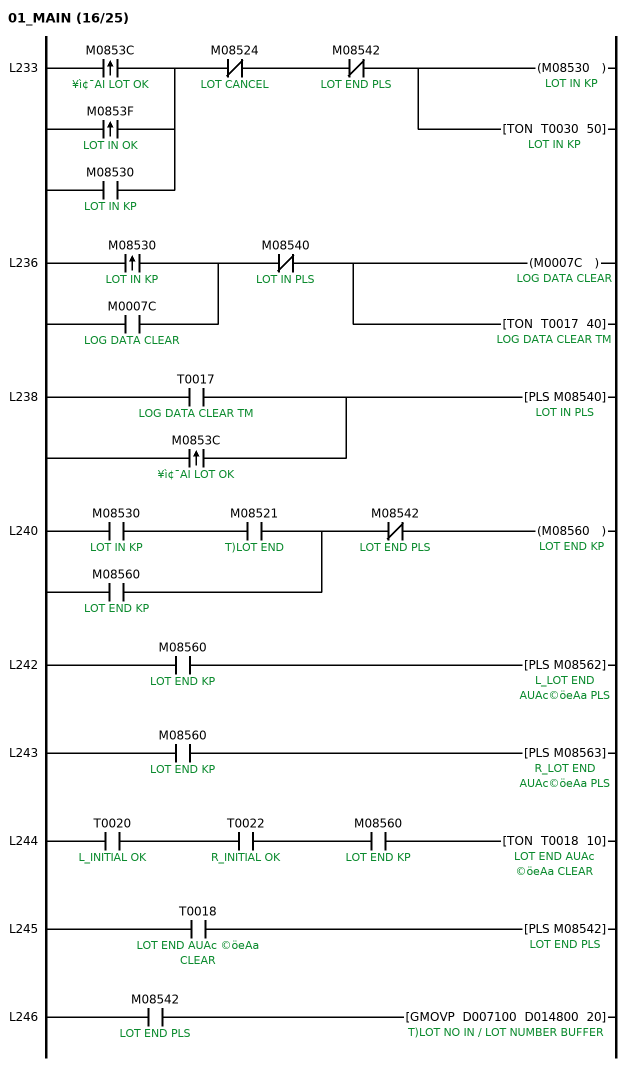
; L233
LOADP     M0853C	// ¥ì¢¯AI LOT OK
ORP       M0853F	// LOT IN OK
OR        M08530	// LOT IN KP
AND NOT   M08524	// LOT CANCEL
AND NOT   M08542	// LOT END PLS
OUT       M08530	// LOT IN KP
TON       T0030 50	// LOT IN KP
; L236
LOADP     M08530	// LOT IN KP
OR        M0007C	// LOG DATA CLEAR
AND NOT   M08540	// LOT IN PLS
OUT       M0007C	// LOG DATA CLEAR
TON       T0017 40	// LOG DATA CLEAR TM
; L238
LOAD      T0017	// LOG DATA CLEAR TM
ORP       M0853C	// ¥ì¢¯AI LOT OK
OUTP      M08540	// LOT IN PLS
; L240
LOAD      M08530	// LOT IN KP
AND       M08521	// T)LOT END
OR        M08560	// LOT END KP
AND NOT   M08542	// LOT END PLS
OUT       M08560	// LOT END KP
; L242
LOAD      M08560	// LOT END KP
OUTP      M08562	// L_LOT END AUAc©öeAa PLS
; L243
LOAD      M08560	// LOT END KP
OUTP      M08563	// R_LOT END AUAc©öeAa PLS
; L244
LOAD      T0020	// L_INITIAL OK
AND       T0022	// R_INITIAL OK
AND       M08560	// LOT END KP
TON       T0018 10	// LOT END AUAc ©öeAa CLEAR
; L245
LOAD      T0018	// LOT END AUAc ©öeAa CLEAR
OUTP      M08542	// LOT END PLS
; L246
LOAD      M08542	// LOT END PLS
GMOVP     D007100 D014800 20	// T)LOT NO IN / LOT NUMBER BUFFER

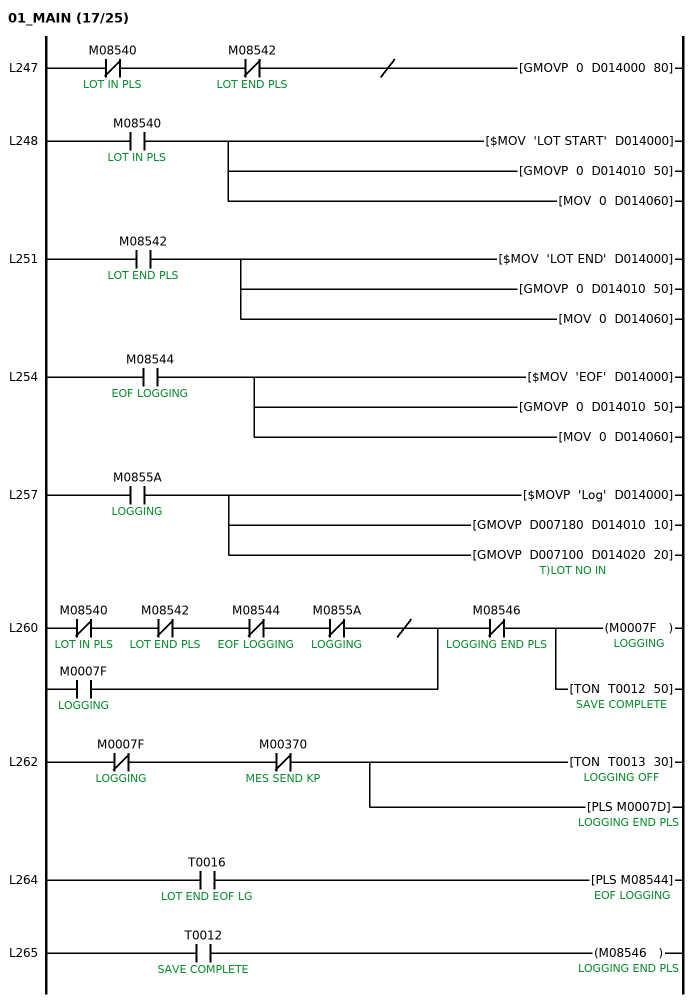
; L247
LOAD NOT  M08540	// LOT IN PLS
AND NOT   M08542	// LOT END PLS
NOT
GMOVP     0 D014000 80
; L248
LOAD      M08540	// LOT IN PLS
$MOV      'LOT START' D014000
GMOVP     0 D014010 50
MOV       0 D014060
; L251
LOAD      M08542	// LOT END PLS
$MOV      'LOT END' D014000
GMOVP     0 D014010 50
MOV       0 D014060
; L254
LOAD      M08544	// EOF LOGGING
$MOV      'EOF' D014000
GMOVP     0 D014010 50
MOV       0 D014060
; L257
LOAD      M0855A	// LOGGING
$MOVP     'Log' D014000
GMOVP     D007180 D014010 10
GMOVP     D007100 D014020 20	// T)LOT NO IN
; L260
LOAD NOT  M08540	// LOT IN PLS
AND NOT   M08542	// LOT END PLS
AND NOT   M08544	// EOF LOGGING
AND NOT   M0855A	// LOGGING
NOT
OR        M0007F	// LOGGING
AND NOT   M08546	// LOGGING END PLS
OUT       M0007F	// LOGGING
TON       T0012 50	// SAVE COMPLETE
; L262
LOAD NOT  M0007F	// LOGGING
AND NOT   M00370	// MES SEND KP
TON       T0013 30	// LOGGING OFF
OUTP      M0007D	// LOGGING END PLS
; L264
LOAD      T0016	// LOT END EOF LG
OUTP      M08544	// EOF LOGGING
; L265
LOAD      T0012	// SAVE COMPLETE
OUT       M08546	// LOGGING END PLS

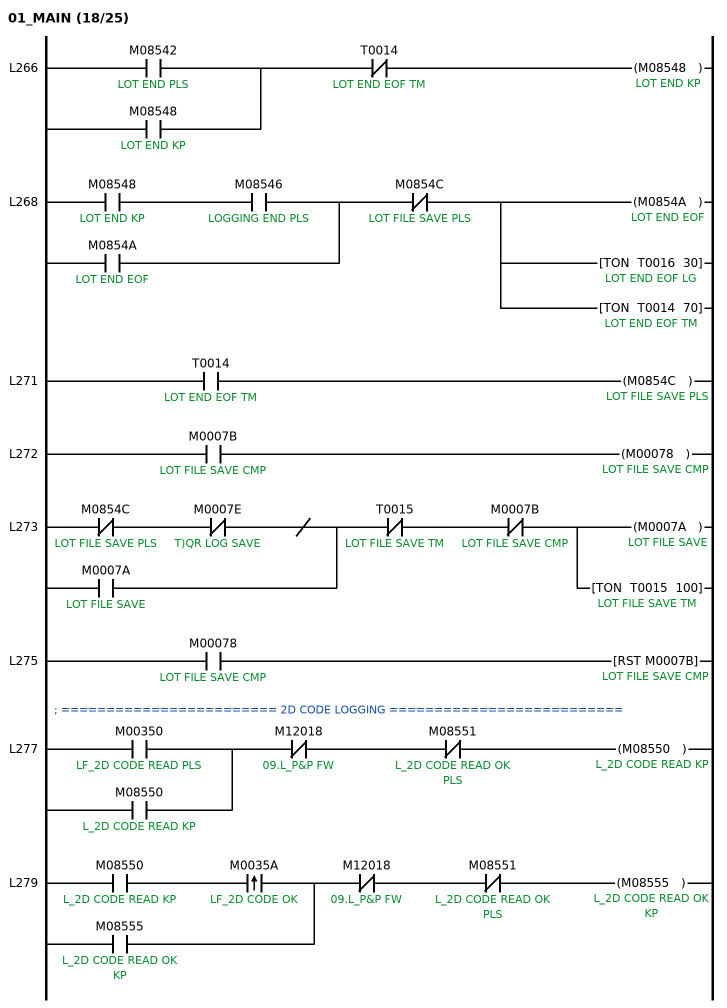
; L266
LOAD      M08542	// LOT END PLS
OR        M08548	// LOT END KP
AND NOT   T0014	// LOT END EOF TM
OUT       M08548	// LOT END KP
; L268
LOAD      M08548	// LOT END KP
AND       M08546	// LOGGING END PLS
OR        M0854A	// LOT END EOF
AND NOT   M0854C	// LOT FILE SAVE PLS
OUT       M0854A	// LOT END EOF
TON       T0016 30	// LOT END EOF LG
TON       T0014 70	// LOT END EOF TM
; L271
LOAD      T0014	// LOT END EOF TM
OUT       M0854C	// LOT FILE SAVE PLS
; L272
LOAD      M0007B	// LOT FILE SAVE CMP
OUT       M00078	// LOT FILE SAVE CMP
; L273
LOAD NOT  M0854C	// LOT FILE SAVE PLS
AND NOT   M0007E	// T)QR LOG SAVE
NOT
OR        M0007A	// LOT FILE SAVE
AND NOT   T0015	// LOT FILE SAVE TM
AND NOT   M0007B	// LOT FILE SAVE CMP
OUT       M0007A	// LOT FILE SAVE
TON       T0015 100	// LOT FILE SAVE TM
; L275
LOAD      M00078	// LOT FILE SAVE CMP
RST       M0007B	// LOT FILE SAVE CMP
// ======================== 2D CODE LOGGING ==========================
; L277
LOAD      M00350	// LF_2D CODE READ PLS
OR        M08550	// L_2D CODE READ KP
AND NOT   M12018	// 09.L_P&P FW
AND NOT   M08551	// L_2D CODE READ OK PLS
OUT       M08550	// L_2D CODE READ KP
; L279
LOAD      M08550	// L_2D CODE READ KP
ANDP      M0035A	// LF_2D CODE OK
OR        M08555	// L_2D CODE READ OK KP
AND NOT   M12018	// 09.L_P&P FW
AND NOT   M08551	// L_2D CODE READ OK PLS
OUT       M08555	// L_2D CODE READ OK KP

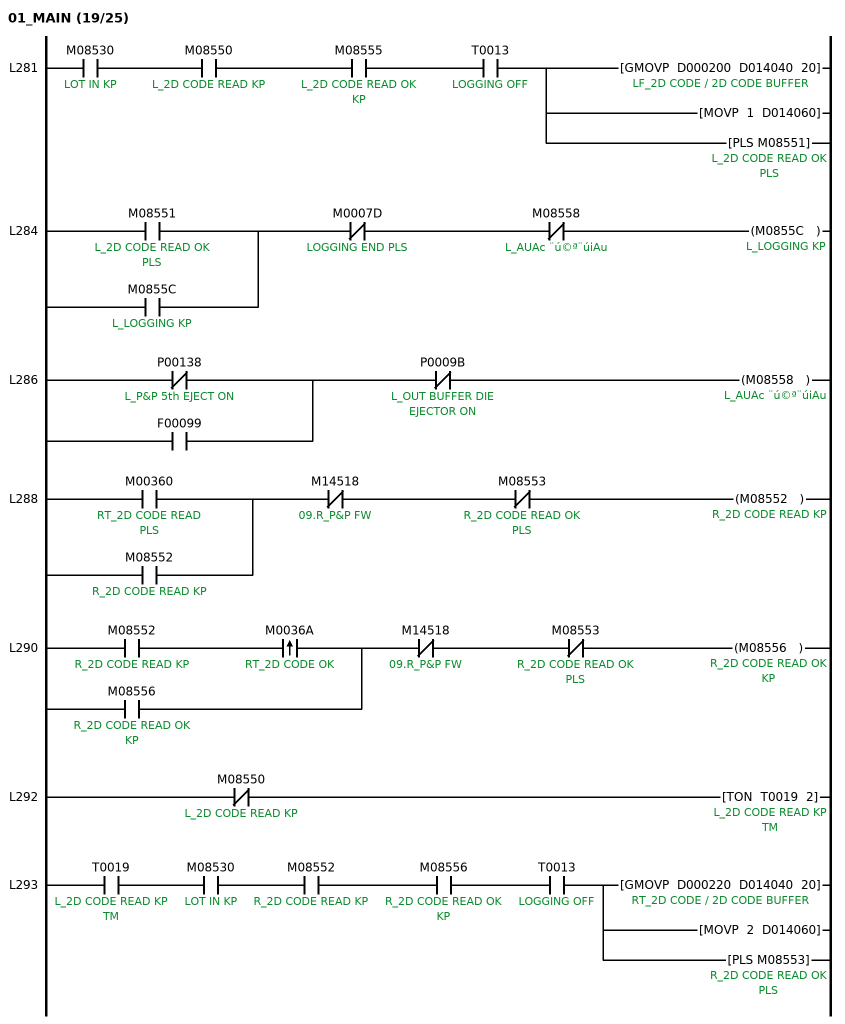
; L281
LOAD      M08530	// LOT IN KP
AND       M08550	// L_2D CODE READ KP
AND       M08555	// L_2D CODE READ OK KP
AND       T0013	// LOGGING OFF
GMOVP     D000200 D014040 20	// LF_2D CODE / 2D CODE BUFFER
MOVP      1 D014060
OUTP      M08551	// L_2D CODE READ OK PLS
; L284
LOAD      M08551	// L_2D CODE READ OK PLS
OR        M0855C	// L_LOGGING KP
AND NOT   M0007D	// LOGGING END PLS
AND NOT   M08558	// L_AUAc ¨ú©ª¨úiAu
OUT       M0855C	// L_LOGGING KP
; L286
LOAD NOT  P00138	// L_P&P 5th EJECT ON
OR        F00099
AND NOT   P0009B	// L_OUT BUFFER DIE EJECTOR ON
OUT       M08558	// L_AUAc ¨ú©ª¨úiAu
; L288
LOAD      M00360	// RT_2D CODE READ PLS
OR        M08552	// R_2D CODE READ KP
AND NOT   M14518	// 09.R_P&P FW
AND NOT   M08553	// R_2D CODE READ OK PLS
OUT       M08552	// R_2D CODE READ KP
; L290
LOAD      M08552	// R_2D CODE READ KP
ANDP      M0036A	// RT_2D CODE OK
OR        M08556	// R_2D CODE READ OK KP
AND NOT   M14518	// 09.R_P&P FW
AND NOT   M08553	// R_2D CODE READ OK PLS
OUT       M08556	// R_2D CODE READ OK KP
; L292
LOAD NOT  M08550	// L_2D CODE READ KP
TON       T0019 2	// L_2D CODE READ KP TM
; L293
LOAD      T0019	// L_2D CODE READ KP TM
AND       M08530	// LOT IN KP
AND       M08552	// R_2D CODE READ KP
AND       M08556	// R_2D CODE READ OK KP
AND       T0013	// LOGGING OFF
GMOVP     D000220 D014040 20	// RT_2D CODE / 2D CODE BUFFER
MOVP      2 D014060
OUTP      M08553	// R_2D CODE READ OK PLS

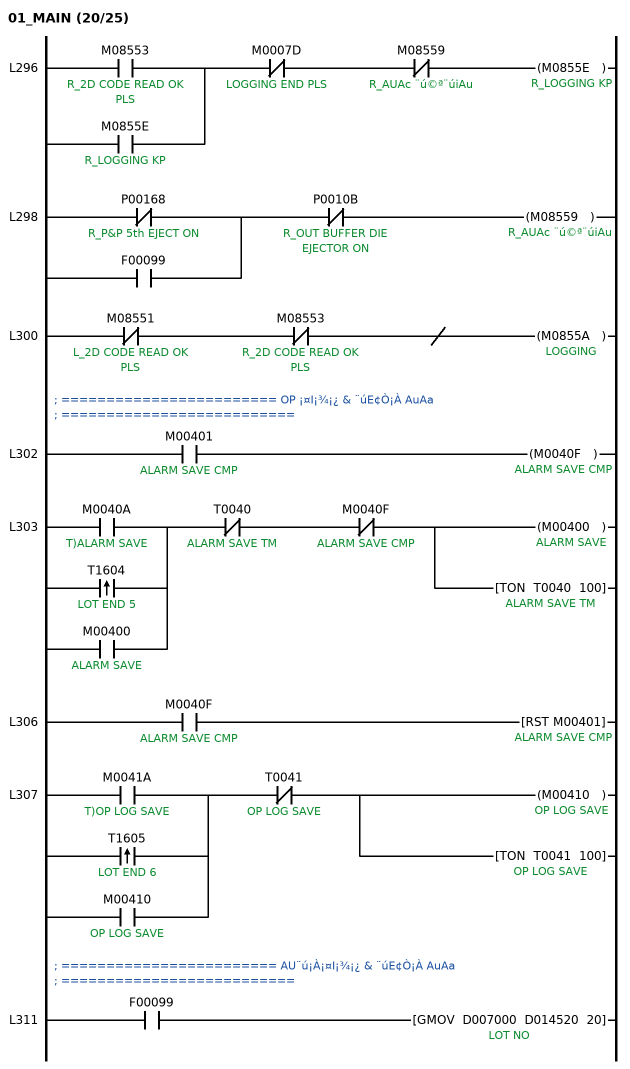
; L296
LOAD      M08553	// R_2D CODE READ OK PLS
OR        M0855E	// R_LOGGING KP
AND NOT   M0007D	// LOGGING END PLS
AND NOT   M08559	// R_AUAc ¨ú©ª¨úiAu
OUT       M0855E	// R_LOGGING KP
; L298
LOAD NOT  P00168	// R_P&P 5th EJECT ON
OR        F00099
AND NOT   P0010B	// R_OUT BUFFER DIE EJECTOR ON
OUT       M08559	// R_AUAc ¨ú©ª¨úiAu
; L300
LOAD NOT  M08551	// L_2D CODE READ OK PLS
AND NOT   M08553	// R_2D CODE READ OK PLS
NOT
OUT       M0855A	// LOGGING
// ======================== OP ¡¤I¡¾¡¿ & ¨úE¢Ò¡À AuAa ==========================
; L302
LOAD      M00401	// ALARM SAVE CMP
OUT       M0040F	// ALARM SAVE CMP
; L303
LOAD      M0040A	// T)ALARM SAVE
ORP       T1604	// LOT END 5
OR        M00400	// ALARM SAVE
AND NOT   T0040	// ALARM SAVE TM
AND NOT   M0040F	// ALARM SAVE CMP
OUT       M00400	// ALARM SAVE
TON       T0040 100	// ALARM SAVE TM
; L306
LOAD      M0040F	// ALARM SAVE CMP
RST       M00401	// ALARM SAVE CMP
; L307
LOAD      M0041A	// T)OP LOG SAVE
ORP       T1605	// LOT END 6
OR        M00410	// OP LOG SAVE
AND NOT   T0041	// OP LOG SAVE
OUT       M00410	// OP LOG SAVE
TON       T0041 100	// OP LOG SAVE
// ======================== AU¨ú¡À¡¤I¡¾¡¿ & ¨úE¢Ò¡À AuAa ==========================
; L311
LOAD      F00099
GMOV      D007000 D014520 20	// LOT NO

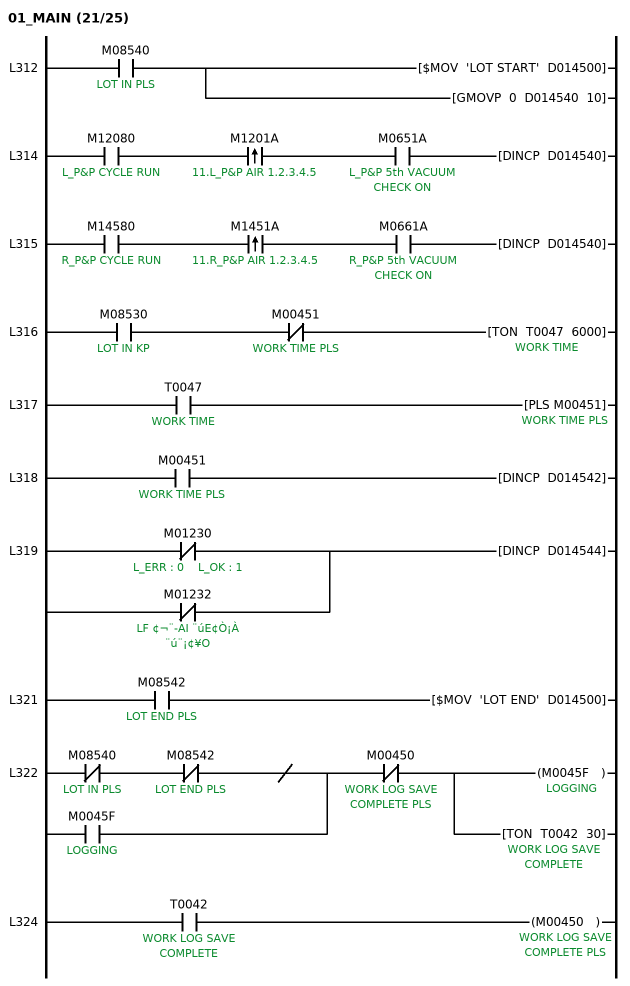
; L312
LOAD      M08540	// LOT IN PLS
$MOV      'LOT START' D014500
GMOVP     0 D014540 10
; L314
LOAD      M12080	// L_P&P CYCLE RUN
ANDP      M1201A	// 11.L_P&P AIR 1.2.3.4.5
AND       M0651A	// L_P&P 5th VACUUM CHECK ON
DINCP     D014540
; L315
LOAD      M14580	// R_P&P CYCLE RUN
ANDP      M1451A	// 11.R_P&P AIR 1.2.3.4.5
AND       M0661A	// R_P&P 5th VACUUM CHECK ON
DINCP     D014540
; L316
LOAD      M08530	// LOT IN KP
AND NOT   M00451	// WORK TIME PLS
TON       T0047 6000	// WORK TIME
; L317
LOAD      T0047	// WORK TIME
OUTP      M00451	// WORK TIME PLS
; L318
LOAD      M00451	// WORK TIME PLS
DINCP     D014542
; L319
LOAD NOT  M01230	// L_ERR : 0    L_OK : 1
OR NOT    M01232	// LF ¢¬¨­AI ¨úE¢Ò¡À ¨ú¨¡¢¥O
DINCP     D014544
; L321
LOAD      M08542	// LOT END PLS
$MOV      'LOT END' D014500
; L322
LOAD NOT  M08540	// LOT IN PLS
AND NOT   M08542	// LOT END PLS
NOT
OR        M0045F	// LOGGING
AND NOT   M00450	// WORK LOG SAVE COMPLETE PLS
OUT       M0045F	// LOGGING
TON       T0042 30	// WORK LOG SAVE COMPLETE
; L324
LOAD      T0042	// WORK LOG SAVE COMPLETE
OUT       M00450	// WORK LOG SAVE COMPLETE PLS

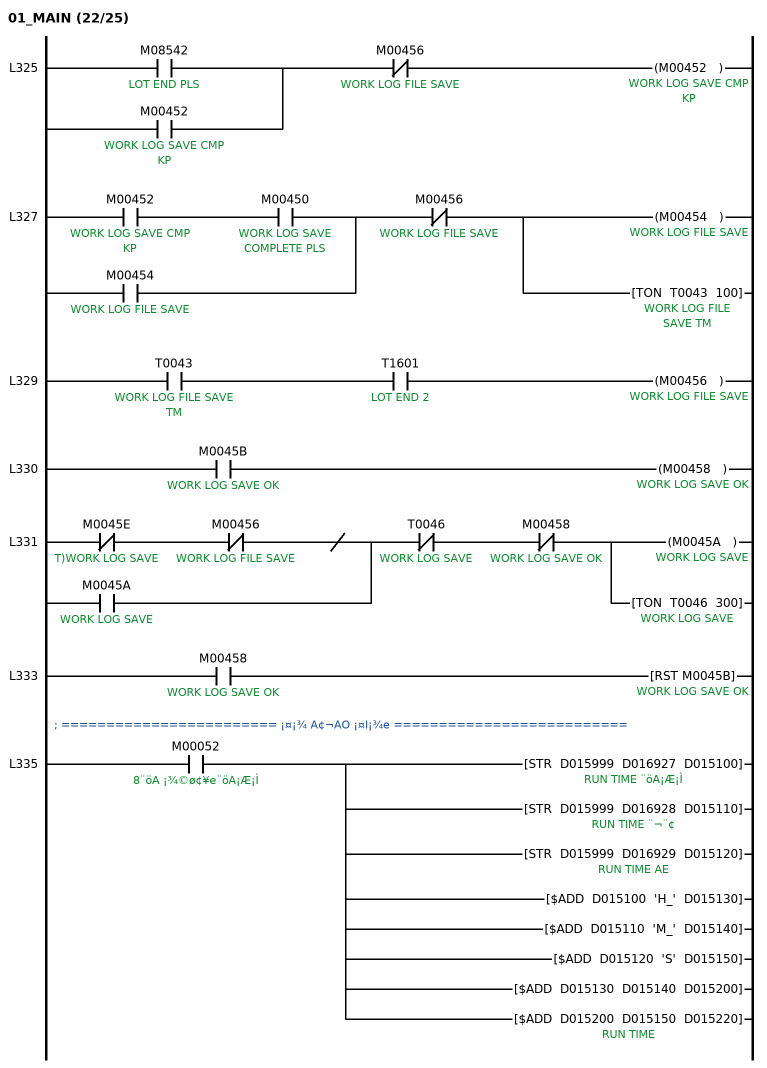
; L325
LOAD      M08542	// LOT END PLS
OR        M00452	// WORK LOG SAVE CMP KP
AND NOT   M00456	// WORK LOG FILE SAVE
OUT       M00452	// WORK LOG SAVE CMP KP
; L327
LOAD      M00452	// WORK LOG SAVE CMP KP
AND       M00450	// WORK LOG SAVE COMPLETE PLS
OR        M00454	// WORK LOG FILE SAVE
AND NOT   M00456	// WORK LOG FILE SAVE
OUT       M00454	// WORK LOG FILE SAVE
TON       T0043 100	// WORK LOG FILE SAVE TM
; L329
LOAD      T0043	// WORK LOG FILE SAVE TM
AND       T1601	// LOT END 2
OUT       M00456	// WORK LOG FILE SAVE
; L330
LOAD      M0045B	// WORK LOG SAVE OK
OUT       M00458	// WORK LOG SAVE OK
; L331
LOAD NOT  M0045E	// T)WORK LOG SAVE
AND NOT   M00456	// WORK LOG FILE SAVE
NOT
OR        M0045A	// WORK LOG SAVE
AND NOT   T0046	// WORK LOG SAVE
AND NOT   M00458	// WORK LOG SAVE OK
OUT       M0045A	// WORK LOG SAVE
TON       T0046 300	// WORK LOG SAVE
; L333
LOAD      M00458	// WORK LOG SAVE OK
RST       M0045B	// WORK LOG SAVE OK
// ======================== ¡¤¡¾ A¢¬AO ¡¤I¡¾e ==========================
; L335
LOAD      M00052	// 8¨öA ¡¾©ø¢¥e¨öA¡Æ¡Ì
STR       D015999 D016927 D015100	// RUN TIME ¨öA¡Æ¡Ì
STR       D015999 D016928 D015110	// RUN TIME ¨¬¨¢
STR       D015999 D016929 D015120	// RUN TIME AE
$ADD      D015100 'H_' D015130
$ADD      D015110 'M_' D015140
$ADD      D015120 'S' D015150
$ADD      D015130 D015140 D015200
$ADD      D015200 D015150 D015220	// RUN TIME

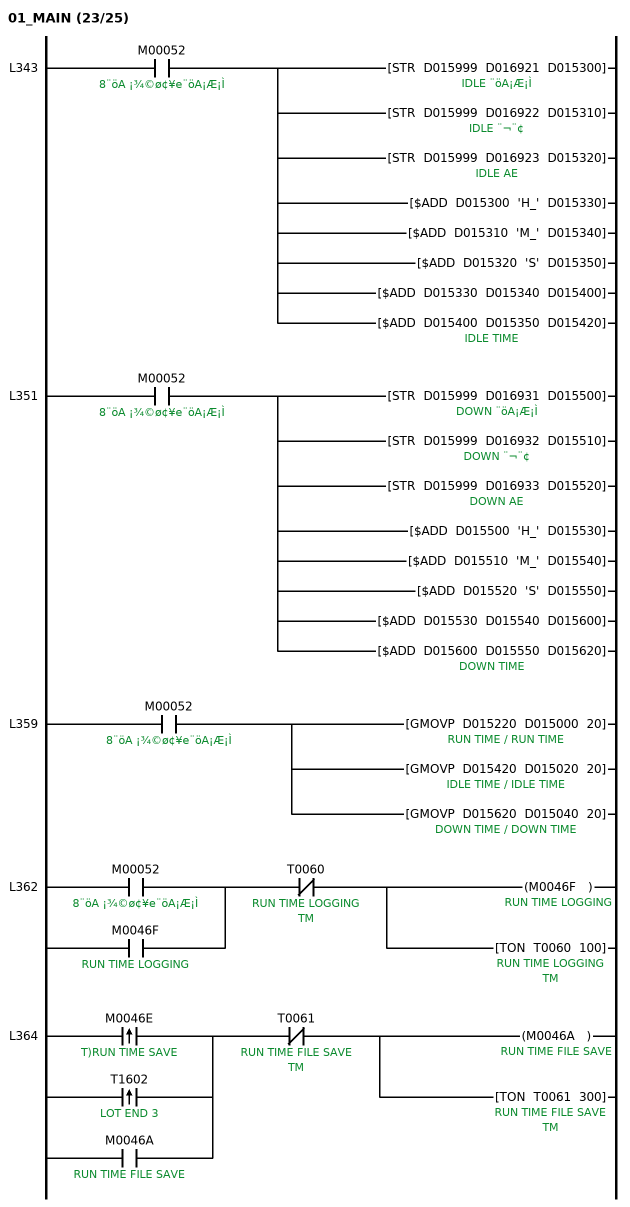
; L343
LOAD      M00052	// 8¨öA ¡¾©ø¢¥e¨öA¡Æ¡Ì
STR       D015999 D016921 D015300	// IDLE ¨öA¡Æ¡Ì
STR       D015999 D016922 D015310	// IDLE ¨¬¨¢
STR       D015999 D016923 D015320	// IDLE AE
$ADD      D015300 'H_' D015330
$ADD      D015310 'M_' D015340
$ADD      D015320 'S' D015350
$ADD      D015330 D015340 D015400
$ADD      D015400 D015350 D015420	// IDLE TIME
; L351
LOAD      M00052	// 8¨öA ¡¾©ø¢¥e¨öA¡Æ¡Ì
STR       D015999 D016931 D015500	// DOWN ¨öA¡Æ¡Ì
STR       D015999 D016932 D015510	// DOWN ¨¬¨¢
STR       D015999 D016933 D015520	// DOWN AE
$ADD      D015500 'H_' D015530
$ADD      D015510 'M_' D015540
$ADD      D015520 'S' D015550
$ADD      D015530 D015540 D015600
$ADD      D015600 D015550 D015620	// DOWN TIME
; L359
LOAD      M00052	// 8¨öA ¡¾©ø¢¥e¨öA¡Æ¡Ì
GMOVP     D015220 D015000 20	// RUN TIME / RUN TIME
GMOVP     D015420 D015020 20	// IDLE TIME / IDLE TIME
GMOVP     D015620 D015040 20	// DOWN TIME / DOWN TIME
; L362
LOAD      M00052	// 8¨öA ¡¾©ø¢¥e¨öA¡Æ¡Ì
OR        M0046F	// RUN TIME LOGGING
AND NOT   T0060	// RUN TIME LOGGING TM
OUT       M0046F	// RUN TIME LOGGING
TON       T0060 100	// RUN TIME LOGGING TM
; L364
LOADP     M0046E	// T)RUN TIME SAVE
ORP       T1602	// LOT END 3
OR        M0046A	// RUN TIME FILE SAVE
AND NOT   T0061	// RUN TIME FILE SAVE TM
OUT       M0046A	// RUN TIME FILE SAVE
TON       T0061 300	// RUN TIME FILE SAVE TM

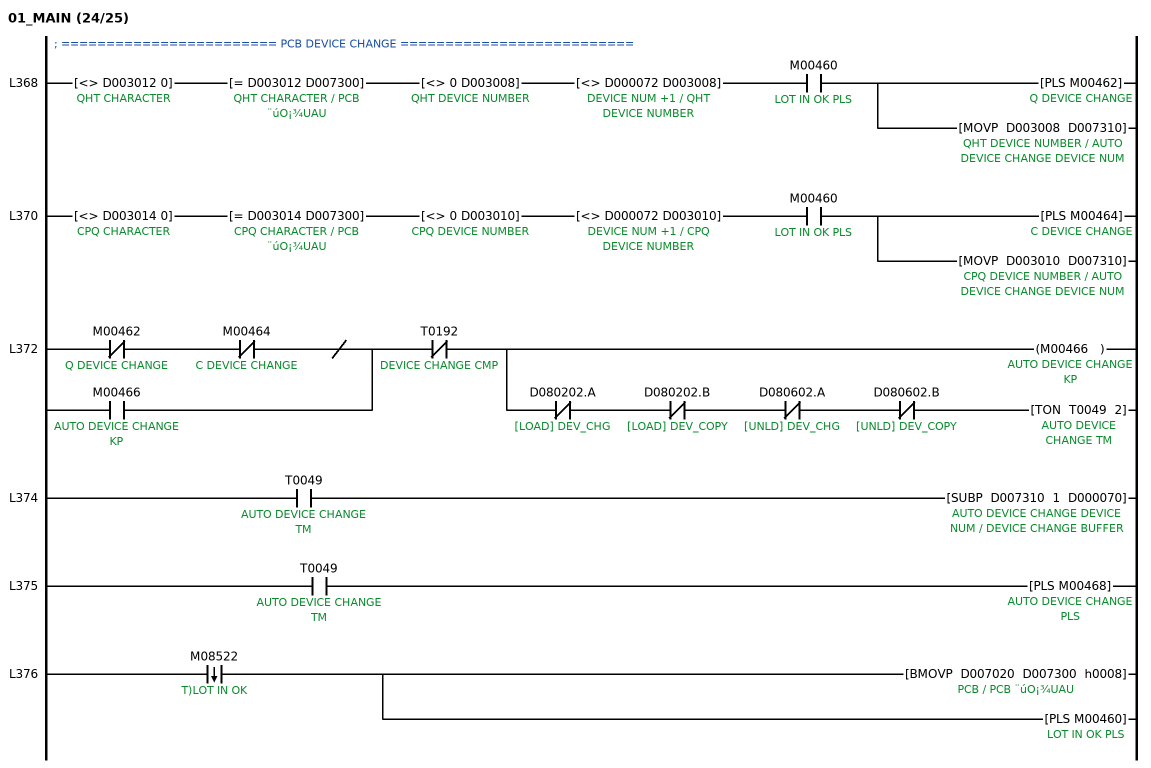
// ======================== PCB DEVICE CHANGE ==========================
; L368
LOAD<>    D003012 0	// QHT CHARACTER
AND=      D003012 D007300	// QHT CHARACTER / PCB ¨úO¡¾UAU
AND<>     0 D003008	// QHT DEVICE NUMBER
AND<>     D000072 D003008	// DEVICE NUM +1 / QHT DEVICE NUMBER
AND       M00460	// LOT IN OK PLS
OUTP      M00462	// Q DEVICE CHANGE
MOVP      D003008 D007310	// QHT DEVICE NUMBER / AUTO DEVICE CHANGE DEVICE NUM
; L370
LOAD<>    D003014 0	// CPQ CHARACTER
AND=      D003014 D007300	// CPQ CHARACTER / PCB ¨úO¡¾UAU
AND<>     0 D003010	// CPQ DEVICE NUMBER
AND<>     D000072 D003010	// DEVICE NUM +1 / CPQ DEVICE NUMBER
AND       M00460	// LOT IN OK PLS
OUTP      M00464	// C DEVICE CHANGE
MOVP      D003010 D007310	// CPQ DEVICE NUMBER / AUTO DEVICE CHANGE DEVICE NUM
; L372
LOAD NOT  M00462	// Q DEVICE CHANGE
AND NOT   M00464	// C DEVICE CHANGE
NOT
OR        M00466	// AUTO DEVICE CHANGE KP
AND NOT   T0192	// DEVICE CHANGE CMP
OUT       M00466	// AUTO DEVICE CHANGE KP
AND NOT   D080202.A	// [LOAD] DEV_CHG
AND NOT   D080202.B	// [LOAD] DEV_COPY
AND NOT   D080602.A	// [UNLD] DEV_CHG
AND NOT   D080602.B	// [UNLD] DEV_COPY
TON       T0049 2	// AUTO DEVICE CHANGE TM
; L374
LOAD      T0049	// AUTO DEVICE CHANGE TM
SUBP      D007310 1 D000070	// AUTO DEVICE CHANGE DEVICE NUM / DEVICE CHANGE BUFFER
; L375
LOAD      T0049	// AUTO DEVICE CHANGE TM
OUTP      M00468	// AUTO DEVICE CHANGE PLS
; L376
LOADN     M08522	// T)LOT IN OK
BMOVP     D007020 D007300 h0008	// PCB / PCB ¨úO¡¾UAU
OUTP      M00460	// LOT IN OK PLS

